# B&R Automation Studio project MIG1 (part 8)

#### UDP_Client.c - Init, cyclic, exit code
```c
#include <bur/plctypes.h>

#ifdef _DEFAULT_INCLUDES
	#include <AsDefault.h>
#endif
#include <..\GlobalDef.h>
#include <..\GlobalDecl.h>

#include <..\Lib\Statelib.c>
#include <..\Lib\LoggerLib.c>
#include <..\Lib\WSI_lib.c>

_LOCAL char TML_PLC_IP_Address[16];

typedef struct UDP_int_typ{

	UdpSend_typ send;
	UdpRecv_typ receive;
	UdpClose_typ close;
	UdpOpen_typ	open;

}UDP_int_typ;

typedef struct UDP_typ{

    UINT Step;

	UDINT SentCntr;
	UDINT RecevCntr;

	UDP_int_typ Intr;
	RS_Channel_typ *pSendChan;
	RS_Channel_typ *pRecevChan;

}UDP_typ;

_LOCAL UDP_typ UDP_Config[2];
_LOCAL UDP_typ UDP_Msg[2];

_LOCAL plcstring SrvIP[20];

_LOCAL UINT status;
_LOCAL plcbit sendNewMsg;
_LOCAL UINT receive_cntr;
_LOCAL UINT push_Cntr;

_LOCAL UINT ReceivedCntr;

_LOCAL plcstring KK_String[128];
_LOCAL USINT KK_Char;

_LOCAL plcbit firstScan;

void _INIT ProgramInit(void)
{UINT i;

	strcpy(SrvIP , "192.168.10.11");  // Must be Axis ID 10
	//strcpy(SrvIP , "192.168.19.11"); // This is default IP in new converter
	//strcpy(SrvIP , "255.255.255.255");

	//strcpy(TML_PLC_IP_Address , "192.168.11.123" ); // My PLC  Address - PowerLink Channel
	strcpy(TML_PLC_IP_Address , "192.168.10.123" ); // My PLC  Address - Ethernet Channel

	i = 0;
	// Initialize UDP open function block
	UDP_Config[i].Intr.open.enable = 0;
	UDP_Config[i].Intr.open.options = 0;
	UDP_Config[i].Intr.open.pIfAddr = (UDINT)&TML_PLC_IP_Address[0];
	UDP_Config[i].Intr.open.port = 30689;
	UDP_Config[i].Intr.open.ident = 0;

	// Initialize UDP send function block
	UDP_Config[i].Intr.send.enable = 0;
	UDP_Config[i].Intr.send.flags = 0;
	UDP_Config[i].Intr.send.pHost = (UDINT)&SrvIP[0];
	UDP_Config[i].Intr.send.port = 30689;

	UDP_Config[i].Intr.receive.ident = 0;
	UDP_Config[i].Intr.receive.enable = 1;
	UDP_Config[i].Intr.receive.pIpAddr = 0;
	UDP_Config[i].Intr.receive.flags = 0;

	// Initialize UDP open function block
	UDP_Msg[i].Intr.open.enable = 0;
	UDP_Msg[i].Intr.open.options = 0;
	UDP_Msg[i].Intr.open.pIfAddr = (UDINT)&TML_PLC_IP_Address[0];
	UDP_Msg[i].Intr.open.port = 1700;
	UDP_Msg[i].Intr.open.ident = 0;

	// Initialize UDP send function block
	UDP_Msg[i].Intr.send.enable = 0;
	UDP_Msg[i].Intr.send.flags = 0;
	UDP_Msg[i].Intr.send.pHost = (UDINT)&SrvIP[0];
	UDP_Msg[i].Intr.send.port = 1700;

	UDP_Msg[i].Intr.receive.ident = 0;
	UDP_Msg[i].Intr.receive.enable = 1;
	UDP_Msg[i].Intr.receive.flags = 0;
	UDP_Msg[i].Intr.receive.pIpAddr = 0;

	////////////////////////////////////////////////////
	UDP_Config[i].pRecevChan = &TML_Data_Chan[1];
	UDP_Config[i].pSendChan = &UDP_Connect_Send[i];

	UDP_Msg[i].pRecevChan = 0;
	UDP_Msg[i].pSendChan = &TML_Msg_Chan[1];

	////////////////////////
	//UDP_Config[i].Step = 1;
	//UDP_Msg[i].Step = 1;

	// Start Connection
	UDP_Config[i].pSendChan->Data[0] = 0x01;
	UDP_Config[i].pSendChan->Len = 1;

	UDP_Ready = 0;

	firstScan = 1;

	//Kick_TML_Cmd = 1;

}

void _CYCLIC ProgramCyclic(void)
{
UINT i , k ;

	//if(ESTOP && firstScan){
	if(firstScan){
		Kick_TML_Cmd = 1;
		firstScan = 0;

	}

	switch(Kick_TML_Cmd){

		case 1:

			UDP_Ready = 0;

			TML_mgr[0].hrdw[0].RXCount = 0;
			TML_mgr[0].hrdw[1].RXCount = 0;

			TML_mgr[1].hrdw[0].RXCount = 0;
			TML_mgr[1].hrdw[1].RXCount = 0;

			TML_mgr[0].hrdw[0].TXCount = 0;
			TML_mgr[0].hrdw[1].TXCount = 0;

			TML_mgr[1].hrdw[0].TXCount = 0;
			TML_mgr[1].hrdw[1].TXCount = 0;

			TML_mgr[0].hrdw[0].TXCountReadBack = TML_mgr[0].hrdw[0].TXCount;
			TML_mgr[0].hrdw[1].TXCountReadBack = TML_mgr[0].hrdw[1].TXCount;

			TML_mgr[1].hrdw[0].TXCountReadBack = TML_mgr[1].hrdw[0].TXCount;
			TML_mgr[1].hrdw[1].TXCountReadBack = TML_mgr[1].hrdw[1].TXCount;

			if(UDP_Config[0].Step == 10)
				UDP_Config[0].Step = 20;
			else
				UDP_Config[0].Step = 1;

			if(UDP_Msg[0].Step == 10)
				UDP_Msg[0].Step = 20;
			else
				UDP_Msg[0].Step = 1;

			Kick_TML_Cmd++;

		break;

		case 2:

			if((UDP_Msg[0].Step == 10)
				&& (UDP_Config[0].Step == 10)){

				UDP_Connect_Send[0].Cntr = 0;
				UDP_Connect_Send[0].Len = 1;

				Kick_TML_Cmd++;

			}

		break;

		case 3:

			if(UDP_Connect_Send[0].Cntr > 0)
				Kick_TML_Cmd++;

			Kick_TML_Cmd++;

		break;

		case 4:

			Kick_TML_Cmd++;

			TML_Msg_Chan[0].Trash_Cntr = 0;
			TML_Data_Chan[0].Trash_Cntr = 0;

			UDP_Ready = 1;

		break;

	}

	for(i = 0 ; i < 1 ; i++){

		for(k = 0 ; k < 2 ; k++){

			switch(k){

				case 0: 	UDP_Socket(&UDP_Config[i]);   	break;

				case 1: 	UDP_Socket(&UDP_Msg[i]);  		break;

			}

		}

	}

}

void UDP_Socket(UDP_typ *udp){

	switch(udp->Step){

			case 0:

			break;

			case 1:

				if(udp->pRecevChan){
					udp->Intr.receive.pData = (UDINT)&udp->pRecevChan->Data[0];
					udp->Intr.receive.datamax = 32;

				}else{
					udp->Intr.receive.pData = 0;
					udp->Intr.receive.datamax = 0;
				}

				if(udp->pSendChan){
					udp->Intr.send.pData = (UDINT)&udp->pSendChan->Data[0];
					udp->Intr.send.datalen = 0;
				}
				else{
					udp->Intr.send.pData = 0;
					udp->Intr.send.datalen = 0;
				}

				udp->Intr.open.enable = 1;

				UdpOpen(&udp->Intr.open);

				if(udp->Intr.open.ident && (udp->Intr.open.status == 0)){

					udp->Intr.send.enable = 1;
					udp->Intr.receive.enable = 1;

					udp->Intr.send.ident = udp->Intr.open.ident;
					udp->Intr.receive.ident = udp->Intr.open.ident;
					udp->Intr.close.ident = udp->Intr.open.ident;

					udp->Step = 10;

				}
				else if(udp->Intr.open.status == 32502){ // Port already opened

					udp->Intr.close.ident = udp->Intr.open.ident;
					udp->Intr.close.enable = 1;
					udp->Step = 20;
				}
				else if(udp->Intr.open.status != ERR_FUB_BUSY)
					udp->Step = 102;

			break;

			case 10:

				//////////////////////////////

				if(udp->pSendChan){

					if(udp->pSendChan->Len > 0){

						udp->Intr.send.datalen = udp->pSendChan->Len;
						UdpSend(&udp->Intr.send);

						if(udp->Intr.send.status == 0){

							udp->Intr.send.datalen = 0;

							udp->pSendChan->_len_prev = udp->pSendChan->Len;
							udp->pSendChan->Len = 0;
							udp->SentCntr++;
							udp->pSendChan->Cntr++;
						}
						else if(udp->Intr.send.status != ERR_FUB_BUSY){

							udp->Intr.send.datalen = 0;

						 	udp->pSendChan->_len_prev = udp->pSendChan->Len;
							udp->pSendChan->Len = 0;
							udp->Step = 110;
						}
					}

				}

				//////////////////////////////////////////////////////////////////

				if(udp->pRecevChan){

					if((udp->pRecevChan->Len == 0)
						&& (udp->pSendChan->Len == 0)){

						UdpRecv(&udp->Intr.receive);

						if(udp->Intr.receive.status == ERR_FUB_BUSY)
						{  }// Process busy

						else if(udp->Intr.receive.status == 0)/* Data received */
						{
							udp->pRecevChan->Len = udp->Intr.receive.recvlen;
							udp->RecevCntr++;
							udp->pRecevChan->Cntr++;

						}
						else if(udp->Intr.receive.status != 32505) // Error ( 32505 is no datat received)
							udp->Step = 115;

					}
				}

			break;

			case 20:

				UdpClose(&udp->Intr.close);

				if(udp->Intr.close.status == ERR_FUB_BUSY)
				{  }// Process busy

				else if(udp->Intr.close.status) {// error
						//udp->Step = 120;
						udp->Step = 1;
				}
				else{

					udp->Intr.open.ident = 0;
					udp->Intr.send.ident = 0;
					udp->Intr.close.ident = 0;
					udp->Intr.receive.ident = 0;

					udp->Step = 1;
				}

			break;

			case 101:
			case 102:
			case 110:
			case 115:
			case 120:

			break;

		}

}
```

### Program Logical/Calibr (ANSIC)

#### Clibr.c - Init, cyclic, exit code
```c
#include <bur/plctypes.h>

#ifdef _DEFAULT_INCLUDES
	#include <AsDefault.h>
#endif

#include <..\GlobalDef.h>
#include <..\GlobalDecl.h>

_LOCAL SINT TVL_Calibr_Cmd;
_LOCAL USINT TVL_Calibr_Step;
_LOCAL TON_typ TVL_Calibr_Tmr;

void _INIT ProgramInit(void)
{

}

void _CYCLIC ProgramCyclic(void)
{

}

void _EXIT ProgramExit(void)
{

}
```

### Program Logical/LincolnPS (ANSIC)

#### LincolnPS.c - Cyclic code
```c
///   ARC Link address: "192.168.10.2"

#include <bur/plctypes.h>

#ifdef _DEFAULT_INCLUDES
	#include <AsDefault.h>
#endif

#include <..\Lib\utilityLib\bgdebug.h>

#include <..\Lib\libUDP\libUDP.h>
#include <..\Lib\libUDP\libUDP.c>

#include <..\Lib\arclink\arclink.h>
#include <..\Lib\arclink\arclink.c>

#define REC_BUF_LEN 	512
#define REC_NUM 	8
#define ARCCOM_TIMEOUT 2000

_GLOBAL Arc_Link_typ ArcLink;

/*
#define REC_BUF_LEN 	4+1
#define REC_NUM 	4
*/

USINT send_data[REC_BUF_LEN];
USINT receive_data[REC_BUF_LEN];
USINT temp_data[REC_BUF_LEN * 3];

_LOCAL RingBuffer RingBufIn;
_LOCAL RingBuffer RingBufOut;
char RingBufInData[(REC_BUF_LEN +4) * REC_NUM];
char RingBufOutData[(REC_BUF_LEN +4) * REC_NUM];
char MsgInData[REC_BUF_LEN];
char MsgOutData[REC_BUF_LEN];

_LOCAL Arc_Link_typ *arcLink;
_LOCAL UDP_typ2 ArcLink_UDP;
_LOCAL plcbit Run_DispatchOutgoingMessages;

_LOCAL char ArcLinkPS_IP_Address[16];
_LOCAL char ArcLinkPLC_IP_Address[16];
_LOCAL plcbit ArcLink_Run;

_LOCAL plcbit KK_ReadParamData;

/*
_LOCAL plcbit RunOutgoingDispatcher;

/// Test Ring Buffer

_LOCAL plcbit KK_Write , KK_Read;
_LOCAL plcstring KK_text_Write[32] ,  KK_text_Read[32];
_LOCAL UDINT KK_Write_Len , KK_Read_Len;
_LOCAL plcbit KK_isEmpty , KK_isFULL;

_LOCAL plcbit K_Send_Req_Action_28 , K_Send_Resp_Action_28;

const char Action_28_Request[29] = {
	0x00, 0x02, 0x0a, 0x4a, 0x00, 0x00, 0x00, 0x00, 0x00, 0x13,
	0x00, 0x32, 0x08, 0x00, 0x00, 0x01, 0x02, 0x01, 0x00, 0x16,
	0x00, 0x00, 0x00, 0xff, 0x01, 0xfe, 0x01, 0x00, 0x01,
};

const char Action_28_Respond[16] = {
	0x00, 0x03, 0x0A, 0x4A, 0x00, 0x00, 0x00, 0x00, 0x00, 0x06,
	0x01, 0x00, 0x00, 0x06, 0x00, 0x00,

};

*/

////////////////////////////////////////////

//UDP Receive Callback function to push data on ring buffer
static void udpReceivedNewData(UDINT pRxBuffer, UDINT RxDataLen , UDINT ringBuf){

	DBG("New Data Received  of Length %d \r\n" , RxDataLen);

	ckConvertByteStreamToHex(pRxBuffer, temp_data, RxDataLen, sizeof(temp_data));
	DBG("(Hex): %s  \r\n" , temp_data);

	if(ringBuf){

		if(!RingBuffer_isFull((RingBuffer*) ringBuf))
			RingBuffer_writeRecord((RingBuffer*) ringBuf, pRxBuffer, RxDataLen);

	}

}
//UDP Transmit Callback function for debugging purpose
static void udpTransmitedNewData(UDINT pTxBuffer, UDINT pTxDataLen){

	DBG("New Data Trasmitted of Length %d  \r\n " , pTxDataLen );
	ckConvertByteStreamToHex(pTxBuffer, temp_data, pTxDataLen, sizeof(temp_data));
	DBG("(Hex): %s  \r\n" , temp_data);

}

//handle network timeout
void ArcLink_Timer(Arc_Link_typ *arc);

//handle error/status interface
void error_status_handler(Arc_Link_typ *arc);

void _INIT ProgramInit(void){
Arc_Link_typ *arc;
UDP_typ2 *udp;

	//ArcLink.robot.Comm.CntrlParamReq.Attribute_ID = 517;
	ArcLink.robot.Comm.CntrlParamReq.Attribute_ID = 0;
	ArcLink.robot.Comm.CntrlParamReq.Weld_Mode = 200;

	/*
	Work-point	517 Primary control.
	Trim	518 Arc length control (typically).
	Wave-Control 1	519 Process adjustment.
	Wave-Control 2	520 Process adjustment.
	Wave-Control 3	521 Process adjustment.
	Wave-Control 4	522 Process adjustment.
	*/

	ArcLink_Run = 1;

	strcpy(ArcLinkPS_IP_Address , "192.168.10.2" );
	//strcpy(ArcLinkPS_IP_Address , "192.168.1.2" ); // Przez PowerLink Module

	strcpy(ArcLinkPLC_IP_Address , "192.168.10.123" ); // My PLC  Address

	Run_DispatchOutgoingMessages = 1;

	udp = &ArcLink_UDP;

	//if(!arcLink)
		//arcLink = ArcLink_init(REC_NUM , REC_BUF_LEN );

	arcLink = &ArcLink;

	if(arcLink){
		udp->listener_config.port = 4323;
		udp->listener_config.buffer = receive_data;
		udp->listener_config.bufferSize = REC_BUF_LEN;
		udp->listener.iRxCallback = (UDINT)udpReceivedNewData;
		//udp->listener.iRxRingBuf = arcLink->bufIN;
		udp->listener.iRxRingBuf = (UDINT)&RingBufIn;

		//strcpy(udp->send.iIPaddress , "192.168.10.2");
		//	strcpy(udp->send.iIPaddress , "192.168.36.88");
		//strcpy(udp->send.iIPaddress , "192.168.10.178");
		udp->send.iPort = 4323;
		udp->send.iBuffer = send_data;
		udp->send.iBufferSize = REC_BUF_LEN;
		udp->send.iTxCallback = (UDINT)udpTransmitedNewData;

		udp->internal.UdpOpen_0.pIfAddr = (UDINT)&ArcLinkPLC_IP_Address[0];

	}
}

void _CYCLIC ProgramCyclic(void){

UDP_typ2 *udp;

	udp = &ArcLink_UDP;

	if(!arcLink)
		return;

	if(!RingBufIn.buffer)
		RingBuffer_Init(&RingBufIn , &RingBufInData , REC_NUM , REC_BUF_LEN);

	if(!RingBufOut.buffer)
		RingBuffer_Init(&RingBufOut , &RingBufOutData , REC_NUM , REC_BUF_LEN);

	if(!arcLink->bufIN
		|| !arcLink->bufOUT
		|| !arcLink->internal.pInMsg
		|| !arcLink->internal.pOutMsg)
	ArcLink_init(arcLink , &RingBufIn, &RingBufOut, MsgInData  , MsgOutData, REC_BUF_LEN );

	//////////////////////////////////////
	if(Run_DispatchOutgoingMessages){

		if(!RingBuffer_isEmpty(arcLink->bufOUT) && !udp->send.iSendCMD){

			udp->send.iBufferSize = RingBuffer_readRecord(arcLink->bufOUT, udp->send.iBuffer);
			udp->send.iSendCMD = 1;

		}

	}

	if((strlen(ArcLinkPS_IP_Address) > 0) && ArcLink_Run) {

		if(udp->internal.step == 0)
			strcpy(udp->send.iIPaddress , ArcLinkPS_IP_Address);

		Udp_cyclic(udp);
		ArcLink_cyclic(arcLink);

	}

	 if(KK_ReadParamData){

	 	KK_ReadParamData = 0;

		ArcLink.robot.Intrf.xCMD = ROBOT_READ_WC_PARAM_DATA;
		ArcLink.robot.Comm.CntrlParamReq.Attribute_ID++;
		if(ArcLink.robot.Comm.CntrlParamReq.Attribute_ID  < 517)
			ArcLink.robot.Comm.CntrlParamReq.Attribute_ID  = 517;
		else if(ArcLink.robot.Comm.CntrlParamReq.Attribute_ID  > 522)
			ArcLink.robot.Comm.CntrlParamReq.Attribute_ID  = 522;

	 }
}
```

### Program Logical/LocalJog (ANSIC)

#### LocalJog.c - Init, cyclic, exit code
```c
#include <bur/plctypes.h>

#ifdef _DEFAULT_INCLUDES
	#include <AsDefault.h>
#endif

#include <..\GlobalDef.h>
#include <..\GlobalDecl.h>

#include <..\Lib\Statelib.c>
#include <..\Lib\LoggerLib.c>
#include <..\Lib\WSI_lib.c>

_LOCAL TON_typ JogMode_Tmr;
_LOCAL float ModeTmo;

_LOCAL plcbit SetLED;

_LOCAL USINT _LocalJogMode;
USINT JogFwdRev(plcbit fwd , plcbit rev);
void LED_Step_Seq();

_LOCAL BOOL blink , _blink;
BOOL _blink;
_LOCAL UINT blinkOnTmr , blinkOffTmr;

_LOCAL TON_typ LED_Tmr;
_LOCAL UINT LED_Indx , LED_Step ;
UINT _LED_Indx;

_LOCAL plcbit LED_Static_Style;

plcbit _Remote_SW;
plcbit _SR_Done;
plcbit _LocalJog_FWD , _LocalJog_REV;

USINT _indx_Limit_Bypass_Btn;

_LOCAL plcbit HMI_INDX_Inp2 , HMI_INDX_Inp3 , HMI_INDX_Out2;

_LOCAL plcbit KK_Block_LED , KK_AllowAll_LED;
_LOCAL float KK_Blink;

void _INIT ProgramInit(void)
{

	KK_Block_LED = 0;
	KK_AllowAll_LED = 0;
	KK_Blink = 0.5;

	Head.Remote_SW = 1;
	ModeTmo = 15.0;

	HardwInit_Done = 0;
	LED_Static_Style = 1;

	Glbl_TML_CMD_Delay = Glbl_TML_CMD_Delay;
}

void _CYCLIC ProgramCyclic(void)
{

USINT tml_indx ;

/*
#define MODE_NONE 	0
#define MODE_TVL 	1
#define MODE_OSC 	2
#define MODE_AHC 	3
#define MODE_WF 	4
#define MODE_INDX 	5

TravelJog.IN
OSCJog_Cmd
AHCJog.IN
WFJog.IN
IndexJog.IN

*/

/** Blink **/
if(blinkOnTmr++ < 150)		blink = 1;
else if(blinkOffTmr++ < 300)	blink = 0;
else{ blinkOnTmr = 0; blinkOffTmr = 0;}

////////////////////////////////////////////////////////
if(HardwReady){

	if(!HardwInit_Done){
		LED_Step = 0;
		LED_CMD = 20;
		_Remote_SW = Head.Remote_SW;
	}

	HardwInit_Done = 1;

}

if(HardwInit_Done && HardwReady){

	Head.Remote_SW = !TML_MTR_INST[TML_AX_WF].DigInp[1];
	//Head.Remote_SW = 1;

	Head.LocalJog_FWD = !TML_MTR_INST[TML_AX_OSC].DigInp[1];
	Head.LocalJog_REV = !TML_MTR_INST[TML_AX_OSC].DigInp[0];

	if(LocalJogMode != MODE_NONE){

		if(Head.LocalJog_FWD || Head.LocalJog_REV)
			TimerStart(&JogMode_Tmr, ModeTmo);

	}

	if((Seq.State > 0) && (Seq.State < 25))
			TimerStart(&JogMode_Tmr, ModeTmo);

	if(!TML_MTR_INST[TML_AX_TVL].DigInp[0]){
		LocalJogMode = MODE_TVL;
		TimerStart(&JogMode_Tmr, ModeTmo);
	}

	else if(!TML_MTR_INST[TML_AX_INDX_EXT].DigInp[1]){
		LocalJogMode = MODE_OSC;
		TimerStart(&JogMode_Tmr, ModeTmo);
	}

	else if(!TML_MTR_INST[TML_AX_TVL].DigInp[1]){
		LocalJogMode = MODE_AHC;
		TimerStart(&JogMode_Tmr, ModeTmo);
	}

	else if(!TML_MTR_INST[TML_AX_INDX].DigInp[1]){
		LocalJogMode = MODE_WF;
		TimerStart(&JogMode_Tmr, ModeTmo);
	}

	else if(!TML_MTR_INST[TML_AX_INDX].DigInp[0] && (!MachCfg.IndxExt)){
		LocalJogMode = MODE_INDX;
		TimerStart(&JogMode_Tmr, ModeTmo);
	}

	else if(!TML_MTR_INST[TML_AX_INDX_EXT].DigInp[0] && (MachCfg.IndxExt)){
		LocalJogMode = MODE_INDX_EXT;
		TimerStart(&JogMode_Tmr, ModeTmo);
	}

	else if(TimerIsTimeOut(&JogMode_Tmr) && (OSC_Step != 10))
		LocalJogMode = MODE_NONE;

}
else {

	Head.Remote_SW = 0;
	Head.LocalJog_FWD = 0;
	Head.LocalJog_REV = 0;

	return;

}

	if(Head.Remote_SW)
		LocalJogMode = MODE_NONE;

	if(Head.Remote_SW && !_Remote_SW)
		//LED_CMD = 40;
		LED_CMD = 10;
	else if(!Head.Remote_SW && _Remote_SW)
		//LED_CMD = 30;
		LED_CMD = 20;

/*
	if(Head.Remote_SW != _Remote_SW){

		OSCJog = Stop;

		OSCJog_Cmd = Stop;

		TravelJog.IN = Stop;

		AHCJog.IN = Stop;

		WFJog.IN = Stop;

		IndexJog.IN = Stop;

	}
	*/

	_Remote_SW = Head.Remote_SW;

//////////  Override POT & NOT on INDX motor

	/*
	if(Head.Remote_SW || !HardwInit_Done || (AccessLevel < 0)){

		INDX_Limit_Bypass_Btn = 0;
		_indx_Limit_Bypass_Btn = INDX_Limit_Bypass_Btn;

	}
	*/

	if(MachCfg.IndxExt)
		tml_indx = TML_AX_INDX_EXT;
	else
		tml_indx = TML_AX_INDX;

	HMI_INDX_Inp2 = TML_MTR_INST[tml_indx].DigInp[2];
	HMI_INDX_Inp3 = TML_MTR_INST[tml_indx].DigInp[3];

	HMI_INDX_Out2 = TML_MTR_INST[tml_indx].DigOut_stat[2];

	if(INDX_Limit_Bypass_Btn && !_indx_Limit_Bypass_Btn){

		if(TML_MTR_INST[tml_indx].xCMD == TML_IDLE){
				TML_MTR_INST[tml_indx].xCMD 	= TML_RST_OUT3_CMD;

			_indx_Limit_Bypass_Btn = INDX_Limit_Bypass_Btn;

		}

	}
	else if(!INDX_Limit_Bypass_Btn && _indx_Limit_Bypass_Btn){

		if(TML_MTR_INST[tml_indx].xCMD == TML_IDLE){
				TML_MTR_INST[tml_indx].xCMD 	= TML_SET_OUT3_CMD;

			_indx_Limit_Bypass_Btn = INDX_Limit_Bypass_Btn;

		}

	}

/////////////////////////////////////////////////////////

	switch(LocalJogMode){

		case MODE_TVL:

			TravelJog.IN = JogFwdRev(Head.LocalJog_FWD , Head.LocalJog_REV);

			if(_LocalJogMode != LocalJogMode)
				LED_CMD = 11;

		break;

		case MODE_OSC:
			 // (0, 1 ,-1)

			if(TML_MTR_INST[TML_AX_INDX_EXT].DigInp[1]){

				if(HardwReady && !Head.Remote_SW){

					if(Head.LocalJog_REV  && !_LocalJog_REV )
						//OSCToggle = 1;
						OSCToggle = !OSCToggle;

					else if(Head.LocalJog_FWD  && !_LocalJog_FWD ){
						if(OSC_Step == 5)
							OSCJog = 1;
						else if(OSC_Step == 10)
							OSCJog = 0;
					}

				}

			}
			else{

				if(Head.LocalJog_FWD == Head.LocalJog_REV)
					OSCJog_Cmd = 0;

				else if(Head.LocalJog_FWD){

					/*
					if(OSCJog)
						OSCJog = 0;
					else */
						OSCJog_Cmd = 1;
				}
				else {
					/*
					if(OSCJog)
						OSCJog = 0;
					else */
						OSCJog_Cmd = -1;
				}
			}

			if(_LocalJogMode != LocalJogMode)
				LED_CMD = 14;

		break;

		case MODE_AHC:

			AHCJog.IN = JogFwdRev(Head.LocalJog_FWD , Head.LocalJog_REV);
			if(_LocalJogMode != LocalJogMode)
				LED_CMD = 13;

		break;

		case MODE_WF:

			WFJog.IN = JogFwdRev(Head.LocalJog_FWD , Head.LocalJog_REV);

			if(_LocalJogMode != LocalJogMode)
				LED_CMD = 15;

		break;

		case MODE_INDX:

			IndexJog.IN = JogFwdRev(Head.LocalJog_FWD , Head.LocalJog_REV);
			if(_LocalJogMode != LocalJogMode)
				LED_CMD = 12;

		break;

		case MODE_INDX_EXT:

			//IndexExtJog.IN = JogFwdRev(Head.LocalJog_FWD , Head.LocalJog_REV);
			IndexJog.IN = JogFwdRev(Head.LocalJog_FWD , Head.LocalJog_REV);
			if(_LocalJogMode != LocalJogMode)
				LED_CMD = 16;

		break;

		default:

			 if (_LocalJogMode != LocalJogMode){

				if(LED_Static_Style)
					LED_CMD = 20;
				else
					LED_CMD = 30;

			 	OSCJog = Stop;

				OSCJog_Cmd = Stop;

				TravelJog.IN = Stop;

				AHCJog.IN = Stop;

				WFJog.IN = Stop;

				IndexJog.IN = Stop;

			}
			 /*
			 else if(HardwReady && !Head.Remote_SW){

				if(Head.LocalJog_FWD && Head.LocalJog_REV && !_LocalJog_FWD_REV )
					OSCToggle = !OSCToggle;

			}
			*/

		break;

	}

	if(_LocalJogMode != LocalJogMode)
		OSCJog = 0;

	_LocalJog_FWD = (Head.LocalJog_FWD);
	_LocalJog_REV = (Head.LocalJog_REV);

	_LocalJogMode = LocalJogMode;
	_blink = blink;
	TimerExecute(&JogMode_Tmr);

	if(LED_CMD){

		TimerStart(&LED_Tmr,0.02);

		if(LED_CMD == 255){ // Reset

			LED_Step = 0;
			LED_Indx = 1;
			LED_CMD = 0;

		}
		else if(LED_CMD <= 10){

			if((LED_Indx > 6)
				|| (LED_Indx == 0))
				LED_Indx = 1;

			LED_Step = LED_CMD;

		}
		else if(LED_CMD < 20){	// Imprtant - Clear & Set

			if((LED_Indx > 6)
			|| (LED_Indx == 0))
				LED_Indx = 1;

			LED_Step = 10;

		}
		else if(LED_CMD == 20){
			LED_Step = 20;
			LED_Indx = 1;
			LED_CMD = 0;

		}
		else if(LED_CMD == 30){
			LED_Step = 30;
			LED_Indx = 1;
			LED_CMD = 0;

		}
		else if(LED_CMD == 40){
			LED_Step = 40;
			LED_Indx = 1;
			LED_CMD = 0;
		}
		else if(LED_CMD == 100){

			if(LED_Step < 100)
				LED_Step = 100;

			LED_CMD = 0;

		}

		else {

			LED_Step = 20;
			LED_CMD = 0;
		}

	}

	if(LED_One_Blink_Req || (Seq.State == 0) || (Seq.State > 25) || KK_AllowAll_LED){

		if(!KK_Block_LED)
			LED_Step_Seq();

	}

	TimerExecute(&LED_Tmr);

}

USINT JogFwdRev(plcbit fwd , plcbit rev){
USINT ret;
// Stop , Reverse , Forward

	if(fwd == rev)
		ret = Stop;
	else if(fwd)
		ret = Forward;
	else if(rev)
		ret = Reverse;
	else
		ret = Stop;

	return ret;

}

void LED_Step_Seq(){

switch(LED_Step){

		case 0:

	/*
	TML_MTR_INST[TML_AX_TVL].xCMD	= TML_SET_OUT1_CMD; // TVL
	TML_MTR_INST[TML_AX_WF].xCMD	= TML_SET_OUT4_CMD; // OUT4 INDX
	TML_MTR_INST[TML_AX_AHC].xCMD	= TML_SET_OUT0_CMD; // AHC
	TML_MTR_INST[TML_AX_OSC].xCMD	= TML_SET_OUT0_CMD; // OSC
	TML_MTR_INST[TML_AX_WF].xCMD	= TML_SET_OUT1_CMD; // WF
	TML_MTR_INST[TML_AX_TVL].xCMD	= TML_SET_OUT4_CMD; // EXT INDX

	TML_SET_OUT1_CMD  		VECT_Rst_OUT1
	*/

		break;

		//////////////////////////////////////////////////////////////////////////////////////

		case 1:

			if(!VectorStateMach[VECT_AX_TVL].xCmd_busy){
				VectorStateMach[VECT_AX_TVL].xCMD 	= VECT_Set_OUT1; // TVL
				LED_CMD = 0;
				LED_Step = 0;

			}
		break;

		case 2:

			if(!VectorStateMach[VECT_AX_WF].xCmd_busy){
				VectorStateMach[VECT_AX_WF].xCMD 	= VECT_Set_OUT4; // OUT4 INDX
				LED_CMD = 0;
				LED_Step = 0;

			}
		break;

		case 3:

			if(!VectorStateMach[VECT_AX_AHC].xCmd_busy){
				VectorStateMach[VECT_AX_AHC].xCMD 	= VECT_Set_OUT0; // AHC
				LED_CMD = 0;
				LED_Step = 0;

			}
		break;

		case 4:

			if(!VectorStateMach[VECT_AX_OSC].xCmd_busy){
				VectorStateMach[VECT_AX_OSC].xCMD 	= VECT_Set_OUT0; // OSC
				LED_CMD = 0;
				LED_Step = 0;

			}
		break;

		case 5:

			if(!VectorStateMach[VECT_AX_WF].xCmd_busy){
				VectorStateMach[VECT_AX_WF].xCMD 	= VECT_Set_OUT1; // WF
				LED_CMD = 0;
				LED_Step = 0;

			}
		break;

		case 6:

			if(!VectorStateMach[VECT_AX_TVL].xCmd_busy){
				VectorStateMach[VECT_AX_TVL].xCMD 	= VECT_Set_OUT4; // EXT INDX
				LED_CMD = 0;
				LED_Step = 0;

			}
		break;

		//****/

		case 10:

			switch(LED_Indx){

				case 1:

					if(!VectorStateMach[VECT_AX_TVL].xCmd_busy){

						VectorStateMach[VECT_AX_TVL].xCMD 	= VECT_Rst_OUT1; // TVL
						//
						LED_Indx++;
					}

				break;

				case 2:

					if(!VectorStateMach[VECT_AX_WF].xCmd_busy){

						VectorStateMach[VECT_AX_WF].xCMD 	= VECT_Rst_OUT4; // OUT4 INDX
						//
						LED_Indx++;
					}

				break;

				case 3:

					if(!VectorStateMach[VECT_AX_AHC].xCmd_busy){
						VectorStateMach[VECT_AX_AHC].xCMD 	= VECT_Rst_OUT0; // AHC
						//
						LED_Indx++;
					}

				break;

				case 4:

					if(!VectorStateMach[VECT_AX_OSC].xCmd_busy){
						VectorStateMach[VECT_AX_OSC].xCMD 	= VECT_Rst_OUT0; // OSC
						//
						LED_Indx++;
					}

				break;

				case 5:

					if(!VectorStateMach[VECT_AX_WF].xCmd_busy){
						VectorStateMach[VECT_AX_WF].xCMD 	= VECT_Rst_OUT1; // WF
						//
						LED_Indx++;
					}

				break;

				case 6:

					if(!VectorStateMach[VECT_AX_TVL].xCmd_busy){
						VectorStateMach[VECT_AX_TVL].xCMD 	= VECT_Rst_OUT4; // EXT INDX
						//
						LED_Indx++;
					}

				break;

				default:

					LED_Indx = 0;

				break;
			}

			if(LED_Indx > 6) {// Done

				if(Head.Remote_SW)
					LED_Step = 40;
				else
					LED_Step = LED_CMD%10;

				LED_CMD = 0;

			}

		break;

		///////////////////////////////////////////////////////////////////////////////

		case 20:

			switch(LED_Indx){

				case 1:

					if(!VectorStateMach[VECT_AX_TVL].xCmd_busy){

						VectorStateMach[VECT_AX_TVL].xCMD 	= VECT_Set_OUT1; // TVL
						//
						LED_Indx++;
					}

				break;

				case 2:

					if(!VectorStateMach[VECT_AX_WF].xCmd_busy){

						VectorStateMach[VECT_AX_WF].xCMD 	= VECT_Set_OUT4; // OUT4 INDX
						//
						LED_Indx++;
					}

				break;

				case 3:

					if(!VectorStateMach[VECT_AX_AHC].xCmd_busy){
						VectorStateMach[VECT_AX_AHC].xCMD 	= VECT_Set_OUT0; // AHC
						//
						LED_Indx++;
					}

				break;

				case 4:

					if(!VectorStateMach[VECT_AX_OSC].xCmd_busy){
						VectorStateMach[VECT_AX_OSC].xCMD 	= VECT_Set_OUT0; // OSC
						//
						LED_Indx++;
					}

				break;

				case 5:

					if(!VectorStateMach[VECT_AX_WF].xCmd_busy){
						VectorStateMach[VECT_AX_WF].xCMD 	= VECT_Set_OUT1; // WF
						//
						LED_Indx++;
					}

				break;

				case 6:

					if(!VectorStateMach[VECT_AX_TVL].xCmd_busy){
						VectorStateMach[VECT_AX_TVL].xCMD 	= VECT_Set_OUT4; // EXT INDX
						//
						LED_Indx++;
					}

				break;

				default:

					LED_Indx = 0;

				break;
			}

			if(LED_Indx > 6){ // Done
				LED_CMD = 0;

				if(LED_Static_Style)
					LED_Step = 0;
				else
					LED_Step = 30;

			}

		break;

		///////////////////////////////////////////////////////////////////////////////

		case 30:

				LED_CMD = 0;
				LED_Indx = 1;
				TimerStart(&LED_Tmr, 0.01);
				_SR_Done = 0;
				LED_Step++;

		break;

		case 31:

			if(LED_CMD)
				LED_Step = 0;

			if(!TimerIsTimeOut(&LED_Tmr))
				break;

			switch(LED_Indx){

				case 1:

					if(!VectorStateMach[VECT_AX_TVL].xCmd_busy){
						VectorStateMach[VECT_AX_TVL].xCMD 	= VECT_Rst_OUT1; // TVL
						_SR_Done = 1;
					}

				break;

				case 2:

					if(!VectorStateMach[VECT_AX_WF].xCmd_busy){
						VectorStateMach[VECT_AX_WF].xCMD 	= VECT_Rst_OUT4; // OUT4 INDX
						_SR_Done = 1;
					}

				break;

				case 3:
					if(!VectorStateMach[VECT_AX_AHC].xCmd_busy){
						VectorStateMach[VECT_AX_AHC].xCMD 	= VECT_Rst_OUT0; // AHC
						_SR_Done = 1;
					}

				break;

				case 4:

					if(!VectorStateMach[VECT_AX_OSC].xCmd_busy){
						VectorStateMach[VECT_AX_OSC].xCMD 	= VECT_Rst_OUT0; // OSC
						_SR_Done = 1;
					}

				break;

				case 5:

					if(!VectorStateMach[VECT_AX_WF].xCmd_busy){
						VectorStateMach[VECT_AX_WF].xCMD 	= VECT_Rst_OUT1; // WF
						_SR_Done = 1;
					}

				break;

				case 6:

					if(!VectorStateMach[VECT_AX_TVL].xCmd_busy){
						VectorStateMach[VECT_AX_TVL].xCMD 	= VECT_Rst_OUT4; // EXT INDX
						_SR_Done = 1;
					}

				break;

				default:

					LED_Indx = 0;

				break;
			 }
			if(_SR_Done){
				_SR_Done = 0;
				TimerStart(&LED_Tmr, KK_Blink * 0.5);
				LED_Indx++;
				if(LED_Indx > 6){
					LED_Indx = 1;
					TimerStart(&LED_Tmr, KK_Blink *0.5);
					LED_Step++;
				}

			}

		break;

		case 32:

			if(!TimerIsTimeOut(&LED_Tmr))
				break;

			switch(LED_Indx){

				case 1:
					if(!VectorStateMach[VECT_AX_TVL].xCmd_busy){
						VectorStateMach[VECT_AX_TVL].xCMD 	= VECT_Set_OUT1; // TVL
						_SR_Done = 1;
					}

				break;

				case 2:

					if(!VectorStateMach[VECT_AX_WF].xCmd_busy){
						VectorStateMach[VECT_AX_WF].xCMD 	= VECT_Set_OUT4; // OUT4 INDX
						_SR_Done = 1;
					}

				break;

				case 3:

					if(!VectorStateMach[VECT_AX_AHC].xCmd_busy){
						VectorStateMach[VECT_AX_AHC].xCMD 	= VECT_Set_OUT0; // AHC
						_SR_Done = 1;
					}

				break;

				case 4:

					if(!VectorStateMach[VECT_AX_OSC].xCmd_busy){
						VectorStateMach[VECT_AX_OSC].xCMD 	= VECT_Set_OUT0; // OSC
						_SR_Done = 1;
					}

				break;

				case 5:

					if(!VectorStateMach[VECT_AX_WF].xCmd_busy){
						VectorStateMach[VECT_AX_WF].xCMD 	= VECT_Set_OUT1; // WF
						_SR_Done = 1;
					}

				break;

				case 6:

					if(!VectorStateMach[VECT_AX_TVL].xCmd_busy){
						VectorStateMach[VECT_AX_TVL].xCMD 	= VECT_Set_OUT4; // EXT INDX
						_SR_Done = 1;
					}

				break;

				default:

					LED_Indx = 0;

				break;
			 }

			if(_SR_Done){
				_SR_Done = 0;
				TimerStart(&LED_Tmr, KK_Blink *0.5);
				LED_Indx++;
				if(LED_Indx > 6){
					LED_Indx = 1;
					TimerStart(&LED_Tmr, KK_Blink *0.5);
					LED_Step = 31;
				}

			}

		break;

		case 33:

			if(LED_CMD)
				LED_Step = 0;

			if(!TimerIsTimeOut(&LED_Tmr))
				break;

			switch(LED_Indx){

				case 1:

					if((!VectorStateMach[VECT_AX_TVL].xCmd_busy)){

						VectorStateMach[VECT_AX_TVL].xCMD 	= VECT_Set_OUT1; // TVL
						_SR_Done = 1;
						LED_Indx++;
					}

				break;

				case 2:

					if((!VectorStateMach[VECT_AX_WF].xCmd_busy)){

						VectorStateMach[VECT_AX_WF].xCMD 	= VECT_Set_OUT4; // OUT4 INDX
						_SR_Done = 1;
						LED_Indx++;
					}

				break;

				case 3:

					if((!VectorStateMach[VECT_AX_AHC].xCmd_busy)){
						VectorStateMach[VECT_AX_AHC].xCMD 	= VECT_Set_OUT0; // AHC
						_SR_Done = 1;
						LED_Indx++;
					}

				break;

				case 4:

					if((!VectorStateMach[VECT_AX_OSC].xCmd_busy)){
						VectorStateMach[VECT_AX_OSC].xCMD 	= VECT_Set_OUT0; // OSC
						_SR_Done = 1;
						LED_Indx++;
					}

				break;

				case 5:

					if((!VectorStateMach[VECT_AX_WF].xCmd_busy)){
						VectorStateMach[VECT_AX_WF].xCMD 	= VECT_Set_OUT1; // WF
						_SR_Done = 1;
						LED_Indx++;
					}

				break;

				case 6:

					if((!VectorStateMach[VECT_AX_TVL].xCmd_busy)){
						VectorStateMach[VECT_AX_TVL].xCMD 	= VECT_Set_OUT4; // EXT INDX
						_SR_Done = 1;
						LED_Indx++;
					}

				break;

				default:

					LED_Indx = 0;

				break;
			}

			if(LED_Indx > 6){

				LED_Indx = 1;
			}

			if(_SR_Done){
				_SR_Done = 0;
				TimerStart(&LED_Tmr, KK_Blink *0.5);
				LED_Step = 31;

			}

		break;

		//////////////////////////////////////////////////////////////////////

		case 40:

			LED_CMD = 0;
			LED_Indx = 1;
			TimerStart(&LED_Tmr, 0.1);
			_SR_Done = 0;
			LED_Step++;

		break;

		case 41:

			if(LED_CMD)
				LED_Step = 0;

			if(!TimerIsTimeOut(&LED_Tmr))
				break;

			switch(LED_Indx){

				case 1:

					if(!VectorStateMach[VECT_AX_TVL].xCmd_busy){

						VectorStateMach[VECT_AX_TVL].xCMD	= VECT_Set_OUT1; // TVL
						_SR_Done = 1;
					}

				break;

				case 2:

					if(!VectorStateMach[VECT_AX_WF].xCmd_busy){

						VectorStateMach[VECT_AX_WF].xCMD	= VECT_Set_OUT4; // OUT4 INDX
						_SR_Done = 1;
					}

				break;

				case 3:

					if(!VectorStateMach[VECT_AX_AHC].xCmd_busy){
						VectorStateMach[VECT_AX_AHC].xCMD	= VECT_Set_OUT0; // AHC
						_SR_Done = 1;
					}

				break;

				case 4:

					if(!VectorStateMach[VECT_AX_OSC].xCmd_busy){
						VectorStateMach[VECT_AX_OSC].xCMD	= VECT_Set_OUT0; // OSC
						_SR_Done = 1;
					}

				break;

				case 5:

					if(!VectorStateMach[VECT_AX_WF].xCmd_busy){
						VectorStateMach[VECT_AX_WF].xCMD	= VECT_Set_OUT1; // WF
						_SR_Done = 1;
					}

				break;

				case 6:

					if(!VectorStateMach[VECT_AX_TVL].xCmd_busy){
						VectorStateMach[VECT_AX_TVL].xCMD	= VECT_Set_OUT4; // EXT INDX
						_SR_Done = 1;
					}

				break;

				default:

					LED_Indx = 0;

				break;
			 }
			if(_SR_Done){
				_SR_Done = 0;
				TimerStart(&LED_Tmr, KK_Blink);
				LED_Step++;

			}

		break;

		case 42:

			if(LED_CMD)
				LED_Step = 0;

			if(!TimerIsTimeOut(&LED_Tmr))
				break;

			switch(LED_Indx){

				case 1:

					if(TML_MTR_INST[TML_AX_TVL].Error){

						VectorStateMach[VECT_AX_TVL].xCMD	= VECT_Rst_OUT1; // TVL
						LED_Step = 0;

					}
					else if(!VectorStateMach[VECT_AX_TVL].xCmd_busy){

						VectorStateMach[VECT_AX_TVL].xCMD	= VECT_Rst_OUT1; // TVL
						_SR_Done = 1;
						LED_Indx++;
					}

				break;

				case 2:

					if(TML_MTR_INST[TML_AX_INDX].Error){

						VectorStateMach[VECT_AX_WF].xCMD	= VECT_Rst_OUT4; // OUT4 INDX
						LED_Step = 0;

					}
					else if(!VectorStateMach[VECT_AX_WF].xCmd_busy){

						VectorStateMach[VECT_AX_WF].xCMD	= VECT_Rst_OUT4; // OUT4 INDX
						_SR_Done = 1;
						LED_Indx++;
					}

				break;

				case 3:

					if(TML_MTR_INST[TML_AX_AHC].Error){

						VectorStateMach[VECT_AX_AHC].xCMD	= VECT_Rst_OUT0; // AHC
						LED_Step = 0;

					}
					else if(!VectorStateMach[VECT_AX_AHC].xCmd_busy){
						VectorStateMach[VECT_AX_AHC].xCMD	= VECT_Rst_OUT0; // AHC
						_SR_Done = 1;
						LED_Indx++;
					}

				break;

				case 4:

					if(TML_MTR_INST[TML_AX_OSC].Error){

						VectorStateMach[VECT_AX_OSC].xCMD	= VECT_Rst_OUT0; // OSC
						LED_Step = 0;

					}
					else if(!VectorStateMach[VECT_AX_OSC].xCmd_busy){
						VectorStateMach[VECT_AX_OSC].xCMD	= VECT_Rst_OUT0; // OSC
						_SR_Done = 1;
						LED_Indx++;
					}

				break;

				case 5:

					if(TML_MTR_INST[TML_AX_WF].Error){

						VectorStateMach[VECT_AX_WF].xCMD	= VECT_Rst_OUT1; // WF
						LED_Step = 0;

					}
					else if(!VectorStateMach[VECT_AX_WF].xCmd_busy){
						VectorStateMach[VECT_AX_WF].xCMD	= VECT_Rst_OUT1; // WF
						_SR_Done = 1;
						LED_Indx++;
					}

				break;

				case 6:

					if(TML_MTR_INST[TML_AX_INDX_EXT].Error){

						VectorStateMach[VECT_AX_TVL].xCMD	= VECT_Rst_OUT4; //
						LED_Step = 0;

					}
					else if(TML_MTR_INST[TML_AX_INDX_EXT].xCMD == TML_IDLE){
						VectorStateMach[VECT_AX_TVL].xCMD	= VECT_Rst_OUT4; //
						_SR_Done = 1;
						LED_Indx++;
					}

				break;

				default:

					LED_Indx = 0;

				break;
			}

			if(LED_Indx > 6){

				LED_Indx = 1;

			}

			if(_SR_Done){
				_SR_Done = 0;
				TimerStart(&LED_Tmr, KK_Blink);
				LED_Step = 41;

			}

		break;

		/////////////////////////////////////

		case 100:

			if(LED_CMD != 100){
				LED_Step = 0;
				LED_CMD = 0;
			}

			if(!TimerIsTimeOut(&LED_Tmr))
				break;

			if(LED_Indx == 0)
				LED_Indx = 1;

			switch(LED_Indx){

				case 1:

					if((!VectorStateMach[VECT_AX_TVL].xCmd_busy)
						|| (VectorStateMach[VECT_AX_TVL].xCMD >= VECT_Set_OUT0)){

						VectorStateMach[VECT_AX_TVL].xCMD 	= VECT_Set_OUT1; // TVL
						LED_Indx++;
					}

				break;

				case 2:

					if((!VectorStateMach[VECT_AX_WF].xCmd_busy)
						|| (VectorStateMach[VECT_AX_WF].xCMD >= VECT_Set_OUT0)){

						VectorStateMach[VECT_AX_WF].xCMD 	= VECT_Set_OUT4; // OUT4 INDX
						LED_Indx++;
					}

				break;

				case 3:

					if((!VectorStateMach[VECT_AX_AHC].xCmd_busy)
						|| (VectorStateMach[VECT_AX_AHC].xCMD >= VECT_Set_OUT0)){

						VectorStateMach[VECT_AX_AHC].xCMD 	= VECT_Set_OUT0; // AHC
						LED_Indx++;
					}

				break;

				case 4:

					if((!VectorStateMach[VECT_AX_OSC].xCmd_busy)
						|| (VectorStateMach[VECT_AX_OSC].xCMD >= VECT_Set_OUT0)){

						VectorStateMach[VECT_AX_OSC].xCMD 	= VECT_Set_OUT0; // OSC
						LED_Indx++;
					}

				break;

				case 5:

					if((!VectorStateMach[VECT_AX_WF].xCmd_busy)
						|| (VectorStateMach[VECT_AX_WF].xCMD >= VECT_Set_OUT1)){

						VectorStateMach[VECT_AX_WF].xCMD 	= VECT_Set_OUT0; // WF
						LED_Indx++;
					}

				break;

				case 6:

					if((!VectorStateMach[VECT_AX_TVL].xCmd_busy)
						|| (VectorStateMach[VECT_AX_TVL].xCMD >= VECT_Set_OUT4)){

						VectorStateMach[VECT_AX_TVL].xCMD 	= VECT_Set_OUT4; //
						LED_Indx++;
					}

				break;

				default:

					LED_Indx = 1;

					TimerStart(&LED_Tmr, 0.5);
					LED_Step = 101;

				break;
			}

		break;

		case 101:

			if(LED_CMD != 100){
				LED_Step = 0;
				LED_CMD = 0;
			}

			if(!TimerIsTimeOut(&LED_Tmr))
				break;

			if(LED_Indx == 0)
				LED_Indx = 1;

			switch(LED_Indx){

				case 1:

					if((!VectorStateMach[VECT_AX_TVL].xCmd_busy)
						|| (VectorStateMach[VECT_AX_TVL].xCMD >= VECT_Set_OUT0)){

						VectorStateMach[VECT_AX_TVL].xCMD 	= VECT_Rst_OUT1; // TVL
						LED_Indx++;
					}

				break;

				case 2:

					if((!VectorStateMach[VECT_AX_WF].xCmd_busy)
						|| (VectorStateMach[VECT_AX_WF].xCMD >= VECT_Set_OUT0)){

						VectorStateMach[VECT_AX_WF].xCMD 	= VECT_Rst_OUT4; // OUT4 INDX
						LED_Indx++;
					}

				break;

				case 3:

					if((!VectorStateMach[VECT_AX_AHC].xCmd_busy)
						|| (VectorStateMach[VECT_AX_AHC].xCMD >= VECT_Set_OUT0)){

						VectorStateMach[VECT_AX_AHC].xCMD 	= VECT_Rst_OUT0; // AHC
						LED_Indx++;
					}

				break;

				case 4:

					if((!VectorStateMach[VECT_AX_OSC].xCmd_busy)
						|| (VectorStateMach[VECT_AX_OSC].xCMD >= VECT_Set_OUT0)){

						VectorStateMach[VECT_AX_OSC].xCMD 	= VECT_Rst_OUT0; // OSC
						LED_Indx++;
					}

				break;

				case 5:

					if((!VectorStateMach[VECT_AX_WF].xCmd_busy)
						|| (VectorStateMach[VECT_AX_WF].xCMD >= VECT_Set_OUT1)){

						VectorStateMach[VECT_AX_WF].xCMD 	= VECT_Rst_OUT0; // WF
						LED_Indx++;
					}

				break;

				case 6:

					if((!VectorStateMach[VECT_AX_TVL].xCmd_busy)
						|| (VectorStateMach[VECT_AX_TVL].xCMD >= VECT_Set_OUT4)){

						VectorStateMach[VECT_AX_TVL].xCMD 	= VECT_Rst_OUT4; // EXT INDX
						LED_Indx++;
					}

				break;

				default:

					LED_Indx = 1;

					TimerStart(&LED_Tmr, 1.0);
					LED_Step = 100;

				break;
			}

		break;

	}

if(LED_Indx != _LED_Indx)
	LED_One_Blink_Req = 0;

_LED_Indx = LED_Indx;

return ;
}
```

### Program Logical/Tester (ANSIC)

#### Tester.c - Init, cyclic, exit code
```c
#include <bur/plctypes.h>

#ifdef _DEFAULT_INCLUDES
	#include <AsDefault.h>
#endif

_LOCAL INT MainCounter , CountPeriod , CountDelta , CountPeriod_SP;

INT _mainCounter;

INT Cntr_Incr(INT newVal , INT prevVal );

void _INIT ProgramInit(void)
{

  CountPeriod_SP =	2000;

}

void _CYCLIC ProgramCyclic(void)
{

	if(CountPeriod > CountPeriod_SP){
		CountPeriod = 0;

		CountDelta = Cntr_Incr(MainCounter , _mainCounter);

		_mainCounter = MainCounter;

	}
	else
		CountPeriod++;

	MainCounter--;
}

INT Cntr_Incr(INT newVal , INT prevVal ){
INT ret = 0;

	if(newVal < prevVal)
		return ((0xFFFF - prevVal)+ newVal + 1);
	else
		return (newVal - prevVal);

	return ret;
}
```

### Program Logical/HMI_Report (ANSIC)

#### HMI_Reports.c - Init, cyclic, exit code
```c
#include <bur/plctypes.h>

#ifdef _DEFAULT_INCLUDES
	#include <AsDefault.h>
#endif

//#include <..\Lib\statelib.c>
//#include <..\Lib\xstring.c>

#include <..\GlobalDef.h>
#include <..\GlobalDecl.h>

#include <..\Lib\Statelib.c>
#include <..\Lib\WSI_lib.c>
#include <..\Lib\LoggerLib.c>

#include<HMI_Reports.h>

_GLOBAL UINT Weld_Report_Status , Weld_Report_Start_Enable;

//////////////////////

_LOCAL UINT Page_Step;

_LOCAL DATE_AND_TIME LocalTime;

_LOCAL UINT KK_Catch;
_LOCAL UINT HMI_ClearError_vis;
_LOCAL plcbit HMI_ClearError_btn;

//_LOCAL plcstring KK_str[32] , KK_format[32];
//_LOCAL plcbit KK_CheckString;
//_LOCAL float KK_Float;
_LOCAL SINT KK_Result;
//_LOCAL USINT KK_dzien;

_LOCAL UINT HMI_Lock_Line[16] , HMI_Line_vis[16] , HMI_Ack_Btn_vis[16];
_LOCAL UINT NewFilePage_vis , _NewFilePage_vis , SetTimePage_vis , _SetTimePage_vis;
_LOCAL UINT HMI_Message_Vis;
_LOCAL UINT HMI_Head_Lock;
_LOCAL UINT Ack_Btn[16] , Glb_Ack_Btn , Glb_Ack_Btn_vis;
_LOCAL DTStructure HMI_DTStr;
_LOCAL DTStructure HMI_SetDTStr;
_LOCAL UINT HMI_Encoder_vis;
_LOCAL UINT HMI_InetrpassTemp_upd;
_LOCAL UINT HMI_HeatInput_vis[16] , HMI_PwrRatio_vis[16] , HMI_HeatInputLimit_vis , HMI_PwrRatioLimit_vis;
_LOCAL UINT HMI_UpdateLine;

_LOCAL float Freq , Dwell_In ,Dwell_Out;

//_LOCAL UDINT DwellIn_dec, DwellOut_dec , ExcurTime_dec;
//_LOCAL float _DwellIn, _DwellOut , _ExcurTime;

//  New File Name Data
_LOCAL plcstring HMI_File_BeadLog[16];
_LOCAL plcstring HMI_File_Name[64];
_LOCAL UINT HMI_File_LayerNo , HMI_File_BeadNo;
_LOCAL USINT HMI_File_TempEvery;
_LOCAL float HMI_File_WireDim;
_LOCAL double HMI_PowerRatio;
_LOCAL float HMI_HeatInput;
_LOCAL USINT HMI_PowerRatio_status;
_LOCAL UINT HMI_PowerRatio_Color;

/////////////////////////////
// new in July 2024

_LOCAL UINT HMI_Options_Vis;

///////
_LOCAL UINT GotoScreen , ReadPage , SetPage;

_LOCAL float _PowerRatio , KK_PowerRatio;
_LOCAL UINT LastBad_BEADS_Cnt;

_LOCAL DTSetTime_typ DTSetTime_1;

_LOCAL int _Len[8];

_LOCAL char LongBuf[512];
_LOCAL UDINT LongBufSize;

_LOCAL USINT TempEveryBead_Flag;

UINT _SeqStep;

void  MenuBar();
char* CreateHeaderTxt(char *p);

char* CreateLineTxt(char *p);

SINT IsItNumber(char*p);

float ActTemp();

void _INIT ProgramInit(void)
{
float f;

	//strcpy(KK_str , "80.2");

	strcpy(File_RW2.fileExten , ".txt");
	strcpy(File_RW2.deviceName, "REPORTS");

	//strcpy(KK_format ,"%2d");

	NewFilePage_vis = INVISIBLE;
	SetTimePage_vis = INVISIBLE;

	HMI_Message_Vis = INVISIBLE;

	HMI_Encoder_vis = INVISIBLE;

	HMI_Options_Vis = INVISIBLE;

	_SetTimePage_vis = SetTimePage_vis;

	HMI_PowerRatio_Color = 1;

	TempEveryBead_Flag = 1;

	if(ActTemp() > 340)
		Weld_Report_Status = 4; // Over temprature
	else
		Weld_Report_Status = 3; // Must enter temperature

	LastBad_BEADS_Cnt = Weld_Rep.BEADS_Cnt;

	/*

	if(CurCalib.GenFloatValue[SETUP_FLOAT_POWER_RATIO_LO] < 10.0)
		CurCalib.GenFloatValue[SETUP_FLOAT_POWER_RATIO_LO] = 10.0;

	if(CurCalib.GenFloatValue[SETUP_FLOAT_POWER_RATIO_HI] > 200.0)
		CurCalib.GenFloatValue[SETUP_FLOAT_POWER_RATIO_HI] = 200.0;

	*/

}

void _CYCLIC ProgramCyclic(void)
{
UINT i;
UINT status;
DTGetTime_typ dtGet;
float w1, w2 , f;

dtGet.enable = 1;
DTGetTime(&dtGet);
LocalTime = dtGet.DT1;

//Weld_Rep.Line[Weld_Rep.ActLINE].TimeStamp = dtGet.DT1;

/*

if(KK_CheckString){
	KK_CheckString = 0;

	KK_Result = IsItNumber(KK_str);
	xsprintf(KK_str , KK_format, KK_dzien);

}

if(OSC_TML_Param_Set[0].pDwell_In
	&& OSC_TML_Param_Set[0].pDwell_Out
	&& OSC_TML_Param_Set[0].pFreq){

	_DwellIn = (*OSC_TML_Param_Set[0].pDwell_In);
	_DwellOut = (*OSC_TML_Param_Set[0].pDwell_Out);
	_ExcurTime = (*OSC_TML_Param_Set[0].pFreq);

	DwellIn_dec = (UDINT)(_DwellIn * 10.0 +0.5);
	DwellOut_dec = (UDINT)(_DwellOut * 10.0 +0.5);
	ExcurTime_dec = (UDINT)(_ExcurTime * 10.0 +0.5);

}

*/

if((Weld_Rep.Report_Type == 0)){ // HEAT INPUT

		HMI_HeatInputLimit_vis = VISIBLE;
		HMI_PwrRatioLimit_vis = INVISIBLE;

	for(i = 0 ; i <16 ; i++){
		HMI_HeatInput_vis[i] =  HMI_Line_vis[i];
		HMI_PwrRatio_vis[i] = INVISIBLE;
	}

}
else{

		HMI_PwrRatioLimit_vis = VISIBLE;
		HMI_HeatInputLimit_vis = INVISIBLE;

	for(i = 0 ; i <16 ; i++){
			HMI_PwrRatio_vis[i] =	HMI_Line_vis[i];
			HMI_HeatInput_vis[i] = INVISIBLE;
		}
}

if((Weld_Report_Status < 2) // calculate only when begining and running
	|| HMI_UpdateLine
	|| HMI_InetrpassTemp_upd){ // or when line values are changed

	HMI_UpdateLine = 0;

	Weld_Rep.Line[Weld_Rep.ActLINE].TimeStamp = dtGet.DT1;

	/*

	if(PS_Param_Set[0].pAmpSP)
	  Weld_Rep.Line[Weld_Rep.ActLINE].PrimaryAmps = (*PS_Param_Set[0].pAmpSP);

	if(WIRE_Param_Set[0].pSpeedSp)
	  Weld_Rep.Line[Weld_Rep.ActLINE].PrimaryWireSpeed = (*WIRE_Param_Set[0].pSpeedSp) * 2.3622047244094488188976377952756;

	if(AVC_Param_Set[0].pVoltSP )
	  Weld_Rep.Line[Weld_Rep.ActLINE].PrimaryVolts = (*AVC_Param_Set[0].pVoltSP) ;

	if(OSC_TML_Param_Set[0].pFreq
		&& OSC_TML_Param_Set[0].pDwell_In
		&& OSC_TML_Param_Set[0].pDwell_Out){

		xsprintf(Weld_Rep.Line[Weld_Rep.ActLINE].Dwell_Excursion , "%d - %d - %d" , \
			(UDINT)((*OSC_TML_Param_Set[0].pDwell_In)*10.0 +0.5) , (UDINT)((*OSC_TML_Param_Set[0].pFreq)*10.0 +0.5) , (UDINT)((*OSC_TML_Param_Set[0].pDwell_Out)*10.0 +0.5));
	}

	*/

  	Weld_Rep.Line[Weld_Rep.ActLINE].PrimaryAmps = permMem.Analog_Out[AHCCurrentSPAO_Indx].Value;
  	Weld_Rep.Line[Weld_Rep.ActLINE].PrimaryWireSpeed = permMem.Analog_Out[WireFeedSpeedAO_Indx].Value; //  * 2.3622047244094488188976377952756;
  	Weld_Rep.Line[Weld_Rep.ActLINE].PrimaryVolts = permMem.Analog_Out[ArcVoltsAO_Indx].Value ;

	Freq = permMem.Analog_Out[OSCSpeedAO_Indx].Value;
	Dwell_In = permMem.Analog_Out[OSC_DwellInAO_Indx].Value;
	Dwell_Out = permMem.Analog_Out[OSC_DwellOutAO_Indx].Value;

	xsprintf(Weld_Rep.Line[Weld_Rep.ActLINE].Dwell_Excursion , "%d - %d - %d" , \
		(UDINT)(Dwell_In * 10.0 + 0.5) , (UDINT)( Freq * 10.0 + 0.5) , (UDINT)(Dwell_Out * 10.0 + 0.5));

	if(Weld_Rep.Line[Weld_Rep.ActLINE].Travel_Tungsten > 0.0){
		w1 =  Weld_Rep.Line[Weld_Rep.ActLINE].PrimaryAmps * Weld_Rep.Line[Weld_Rep.ActLINE].PrimaryVolts * 60.0;
			//Weld_Rep.Line[Weld_Rep.ActLINE].HeatInput = (w1/((*TVL_ROT_Param_Set[0].pPrimVel)* 2.3622047244094488188976377952756))*0.001;
		Weld_Rep.Line[Weld_Rep.ActLINE].HeatInput = (w1/Weld_Rep.Line[Weld_Rep.ActLINE].Travel_Tungsten)*0.001;
	}
	else
		Weld_Rep.Line[Weld_Rep.ActLINE].HeatInput = 0.0;

	HMI_HeatInput = Weld_Rep.Line[Weld_Rep.ActLINE].HeatInput;

	if(Weld_Rep.Line[Weld_Rep.ActLINE].Travel_Tungsten > 0.0){

		//w1 =  Weld_Rep.Line[Weld_Rep.ActLINE].PrimaryWireSpeed / (Weld_Rep.Line[Weld_Rep.ActLINE].Travel_Tungsten * 2.3622047244094488188976377952756);
		w1 =  Weld_Rep.Line[Weld_Rep.ActLINE].PrimaryWireSpeed / (Weld_Rep.Line[Weld_Rep.ActLINE].Travel_Tungsten);
		w2 = Weld_Rep.Head.WireDim/2.0;
		w2 = w2*w2 * M_PI;

		if((w1*w2) > 0){

			Weld_Rep.Line[Weld_Rep.ActLINE].PowerRatio = (Weld_Rep.Line[Weld_Rep.ActLINE].PrimaryVolts *Weld_Rep.Line[Weld_Rep.ActLINE].PrimaryAmps)/(w1 * w2)/1000.0;
		}
		else
			Weld_Rep.Line[Weld_Rep.ActLINE].PowerRatio = 0.0;

	}
	else
		Weld_Rep.Line[Weld_Rep.ActLINE].PowerRatio = 0.0;

	HMI_PowerRatio = Weld_Rep.Line[Weld_Rep.ActLINE].PowerRatio;

	//HMI_PowerRatio_status = ((HMI_PowerRatio >= 66.2) &&  (HMI_PowerRatio <= 87.6))? INVISIBLE:VISIBLE;

	Weld_Report_Start_Enable = 0;

	/*
	if((Weld_Rep.Report_Type == 0)){ // HEAT INPUT

		if(HMI_HeatInput < CurCalib.GenFloatValue[SETUP_FLOAT_HEAT_INPUT_LO])
			HMI_PowerRatio_Color = 84;

		else if(HMI_HeatInput > CurCalib.GenFloatValue[SETUP_FLOAT_HEAT_INPUT_HI])
			HMI_PowerRatio_Color = 43;

		else {

			HMI_PowerRatio_Color = 15;
			Weld_Report_Start_Enable = 1;

		}

	}else{

		if(HMI_PowerRatio < CurCalib.GenFloatValue[SETUP_FLOAT_POWER_RATIO_LO])
			HMI_PowerRatio_Color = 84;

		else if(HMI_PowerRatio > CurCalib.GenFloatValue[SETUP_FLOAT_POWER_RATIO_HI])
			HMI_PowerRatio_Color = 43;

		else {

			HMI_PowerRatio_Color = 15;
			Weld_Report_Start_Enable = 1;

		}

	}
	*/

	///* Test Radom
	/*
	if(Master[0].TestMode) // 11 Apr 2022
		Weld_Report_Start_Enable = 1;
	*/

}

else{

	/*
	if(Master[0].TestMode)  ///* Test Radom
		Weld_Report_Start_Enable = 1;
	else
		Weld_Report_Start_Enable = 0;
	*/

	HMI_PowerRatio_Color = 15;

}

/*
switch(CurCalib.GenSetup[SETUP_LOG_OPTION]){

	case 1: // Log After A side

		if(Weld_Report_Status == 2){ // Beat Finished

			if(Master[0].ToolHeadID){

				Weld_Report_Status = 0;
			}

		}

	break;

	case 2: // Log After B side

		if(Weld_Report_Status == 2){ // Beat Finished

			if(!Master[0].ToolHeadID){

				Weld_Report_Status = 0;
			}

		}

	break;

	case 3: // Log After Any Stop - // Allow beat log after any Stop

		if(!Master[0].SeqStep && _SeqStep)
			Weld_Report_Status = 2;

		if(Weld_Report_Status == 2)
			Weld_Report_Start_Enable = 1;

	break;

	default: break;

}

_SeqStep = Master[0].SeqStep;
*/

HMI_PowerRatio_status = (TempEveryBead_Flag > 0 )? VISIBLE:INVISIBLE;

/*

if(HMI_InetrpassTemp_upd){

	if(Weld_Report_Status == 3){ // Must enter temprature

		if(IsItNumber(Weld_Rep.Line[Weld_Rep.ActLINE].InetrpassTemp)>= 0){
			Weld_Report_Status = 0;
			TempEveryBead_Flag = 1;

		}

	}
}

*/

if(HMI_InetrpassTemp_upd){

	HMI_InetrpassTemp_upd = 0;

	if(IsItNumber(Weld_Rep.Line[Weld_Rep.ActLINE].InetrpassTemp)>= 0){

		f = ActTemp();

		if(f > 340.0 ){

			//if(Weld_Report_Status == 0)
				Weld_Report_Status = 4;

		}
		else if( (f < 320.0)  && ( f > 0.0)){

			if(Weld_Report_Status >= 3)
				Weld_Report_Status = 0; // over temperature - no Welding

		}

		if(Weld_Report_Status == 3){ // Must enter temprature

			Weld_Report_Status = 0;
			TempEveryBead_Flag = 1;

		}

		////////////////////

	}

}

if(Weld_Report_Status == 4)
	HMI_PowerRatio_Color = 87;

/////////////////////////
//////////////////

/////////////////////////////////////////////////////////
//Weld_Report_Mode = (CurCalib.GenSetup[SETUP_EXTRAS]&0x1)? 1:0;

//* Test Radom
if((Weld_Report_Status == 2)){
//if((Weld_Report_Status == 2) && !Master[0].TestMode){
 	HMI_Ack_Btn_vis[Weld_Rep.ActLINE] = VISIBLE;
	Glb_Ack_Btn_vis = VISIBLE;
}
else{

	HMI_Ack_Btn_vis[Weld_Rep.ActLINE] = INVISIBLE;
	Glb_Ack_Btn_vis = INVISIBLE;
}

if(NewFilePage_vis == VISIBLE){

	if(_NewFilePage_vis != NewFilePage_vis){

		strcpy(HMI_File_BeadLog , Weld_Rep.Head.WELD_LOG);
		HMI_File_LayerNo =   Weld_Rep.Head.LAYER_No;
		HMI_File_BeadNo = Weld_Rep.Line[0].BeadNo;
		HMI_File_TempEvery = Weld_Rep.Head.TempEvery;
		HMI_File_WireDim = Weld_Rep.Head.WireDim;

	}

	DT_TO_DTStructure(dtGet.DT1, (UDINT) &HMI_DTStr);
	xsprintf(HMI_File_Name, "%s-%d-%d %d-%d-%d %d-%d" , HMI_File_BeadLog , HMI_File_LayerNo , HMI_File_BeadNo , \
							HMI_DTStr.year , HMI_DTStr.month , HMI_DTStr.day , HMI_DTStr.hour , HMI_DTStr.minute);

}
_NewFilePage_vis = NewFilePage_vis;

if(SetTimePage_vis == VISIBLE){

	if(_SetTimePage_vis != SetTimePage_vis)
		DT_TO_DTStructure(LocalTime, (UDINT) &HMI_SetDTStr);

	if(DTSetTime_1.enable){

		DTSetTime_1.DT1 = DTStructure_TO_DT((UDINT) &HMI_SetDTStr);

		DTSetTime(&DTSetTime_1);
		if(!DTSetTime_1.status)
			DTSetTime_1.enable = 0;

		//SetTimePage_vis = INVISIBLE;

	}

}
_SetTimePage_vis = SetTimePage_vis;

////////////////
HMI_ClearError_vis = (File_RW2.Done && File_RW2.Error )? VISIBLE:INVISIBLE;

if(HMI_ClearError_btn){
	HMI_ClearError_btn = 0;

	File_RW2.Error = 0;
	File_RW2.Done = 0;
	File_RW2.CMD = 0;
	Page_Step = 0;

}
////////////////////

switch(Page_Step){

	default:

		GotoScreen = 10;

		if(Weld_Rep.ActLINE < 16 ){

			for (i = Weld_Rep.ActLINE ; i < 16 ; i++){

				HMI_Line_vis[i] = INVISIBLE;
				HMI_Ack_Btn_vis[i] = INVISIBLE;
			}

			for (i = 0 ; i < Weld_Rep.ActLINE ; i++){

					HMI_Line_vis[i] = VISIBLE;
					HMI_Ack_Btn_vis[i] = INVISIBLE;
					HMI_Lock_Line[i] = 1;
			}

		}
		else{

			Weld_Rep.ActLINE = 15;

			for (i = 0 ; i < 15 ; i++){

				HMI_Line_vis[i] = VISIBLE;
				HMI_Ack_Btn_vis[i] = INVISIBLE;
				HMI_Lock_Line[i] = 1;
			}

		}

		HMI_Lock_Line[Weld_Rep.ActLINE] = 0;
		HMI_Ack_Btn_vis[Weld_Rep.ActLINE] = VISIBLE;
		HMI_Line_vis[i] = VISIBLE;

		HMI_Head_Lock = (Weld_Rep.ActLINE > 0)? 1:0;

		HMI_Message_Vis = INVISIBLE;

		Page_Step = 1;

	break;

	case 1:	// Wait for Acknowledge Line

		status = 0;
		for(i = 0 ; i < 16 ; i++){

			if(Ack_Btn[i])
				status = i+1;

		}

		KK_Catch = status;

		if(status > 0 || Glb_Ack_Btn){

			Glb_Ack_Btn = 0;

			for(i = 0 ; i < 16 ; i++)
				Ack_Btn[i] = 0;

			Page_Step = 3;

		}

	break;

	case 3: // Add records TXT

		//NewFilePage_vis = INVISIBLE;

		KK_Result = IsItNumber(Weld_Rep.Line[Weld_Rep.ActLINE].InetrpassTemp);

		_PowerRatio = KK_PowerRatio;

		//status = ((_PowerRatio > 350) || (_PowerRatio < 340))? 1:0;
		//if(status)

		if(KK_Result >= 0){

			f = atof((UDINT) Weld_Rep.Line[Weld_Rep.ActLINE].InetrpassTemp);

			if(f > 340)
				TempEveryBead_Flag = 1;
			else if (f < 300)
				TempEveryBead_Flag = 0;

		}

		//if(HMI_PowerRatio_status == VISIBLE)
			//LastBad_BEADS_Cnt = Weld_Rep.BEADS_Cnt;

		if(TempEveryBead_Flag)
			LastBad_BEADS_Cnt = Weld_Rep.BEADS_Cnt;

		if(((KK_Result< 0))
			&& ((((Weld_Rep.BEADS_Cnt - LastBad_BEADS_Cnt)%(UINT)Weld_Rep.Head.TempEvery) == 0)
				|| (LastBad_BEADS_Cnt == Weld_Rep.BEADS_Cnt))){

			HMI_Message_Vis = VISIBLE;

			Page_Step = 1;

			break;
		}

		strcpy(File_RW2.fileName , Weld_Rep.FileName);
		strcat(File_RW2.fileName , File_RW2.fileExten);
		File_RW2.CMD = F_OPEN_ONLY;

		Page_Step ++;

	break;

	case 4:

		if(File_RW2.Done && !File_RW2.Error){

			if((File_RW2._int.FOpen.filelen == 0)){

				memset(&LongBuf[0] , 0 , 512);
				LongBufSize = 0;

				Weld_Rep.BEADS_Cnt = 1;

				//CreateHeaderTxt(&LongBuf[0]);
				CreateLineTxt(CreateHeaderTxt(LongBuf));

				//File_RW2.pMem = LongBuf;
				//File_RW2.Len = LongBufSize;
				//File_RW2.Offset = 0;

			}
			else{

				for(i = 0 ; i < 512 ; i++)
					LongBuf[i] = 0;

				//memset(&LongBuf[0] , 0 , 512);
				LongBufSize = 0;

				Weld_Rep.BEADS_Cnt++;

				CreateLineTxt(LongBuf);

			}

			File_RW2.pMem = LongBuf;
			File_RW2.Len = LongBufSize;
			File_RW2.Offset = File_RW2._int.FOpen.filelen;

			HMI_Head_Lock = 1;
			File_RW2.CMD = F_WRITE_ONLY;

			Page_Step ++;

		}
		else if(File_RW2.Error){

			//Page_Step = 0;
		}

	break;

	case 5:

		if(File_RW2.Done && !File_RW2.Error ){

			File_RW2.CMD = F_CLOSE_ONLY;

			Page_Step ++;

		}
		else if(File_RW2.Error){

			//Page_Step = 0;
		}

	break;

	case 6:

		if(File_RW2.Done){

			if(File_RW2.Error){

				//Page_Step = 0;

			}else{

				if(Weld_Rep.ActLINE < 15 ){

					HMI_Lock_Line[Weld_Rep.ActLINE] = 1;
					HMI_Ack_Btn_vis[Weld_Rep.ActLINE] = INVISIBLE;
					Weld_Rep.ActLINE++;
					HMI_Line_vis[Weld_Rep.ActLINE] = VISIBLE;
					HMI_Lock_Line[Weld_Rep.ActLINE] = 0;
					HMI_Ack_Btn_vis[Weld_Rep.ActLINE] = VISIBLE;

					i = Weld_Rep.ActLINE;

					memcpy(&Weld_Rep.Line[i] , &Weld_Rep.Line[i-1] , sizeof(Weld_Report_Line_typ));

				}else{

					for(i = 1 ; i < 16 ; i++)
						memcpy(&Weld_Rep.Line[i-1] , &Weld_Rep.Line[i] , sizeof(Weld_Report_Line_typ));

					i = 15;
				}

				Weld_Rep.Line[i].BeadNo = Weld_Rep.Line[i-1].BeadNo + 1;

				if(ActTemp() < 340.0)
				 	strcpy(Weld_Rep.Line[i].InetrpassTemp , "");

				strcpy(Weld_Rep.Line[i].Comments , "");

				if(ActTemp() > 340)
					Weld_Report_Status = 4;
				else
					Weld_Report_Status = 0;

				Page_Step = 1;

			}

		}

	break;

	//////////////////    New Report TXT ////////////////////////////
	 case 80:

		strcpy(Weld_Rep.Head.WELD_LOG , HMI_File_BeadLog);
		Weld_Rep.Head.LAYER_No = HMI_File_LayerNo;
		Weld_Rep.Line[0].BeadNo = HMI_File_BeadNo;
		Weld_Rep.Head.TempEvery = HMI_File_TempEvery;
		Weld_Rep.Head.WireDim = HMI_File_WireDim;
		//'%0.2d'
		DT_TO_DTStructure(dtGet.DT1, (UDINT) &HMI_DTStr);
		xsprintf(Weld_Rep.FileName, "%s-%d-%d %d-%0.2d-%0.2d %0.2d-%0.2d" , Weld_Rep.Head.WELD_LOG , Weld_Rep.Head.LAYER_No , Weld_Rep.Line[0].BeadNo , \
											HMI_DTStr.year , HMI_DTStr.month , HMI_DTStr.day , HMI_DTStr.hour , HMI_DTStr.minute);

		if(Weld_Rep.Head.WireDim <= 0.0)
			Weld_Rep.Head.WireDim = 0.045;

		if(Weld_Rep.Head.TempEvery == 0)
			Weld_Rep.Head.TempEvery = 4;

		i = 0;

		xsprintf(Weld_Rep.Line[i].WelderStamp,"RB 22%d", (DINT)i+1);

		Weld_Rep.Line[i].PrimaryAmps = 100.0;
		Weld_Rep.Line[i].PrimaryWireSpeed = 200.0;
		Weld_Rep.Line[i].PrimaryVolts = 10.0;
		Weld_Rep.Line[i].Travel_Tungsten = 3.0;
		Weld_Rep.Line[i].PowerRatio = 75.0;
		strcpy(Weld_Rep.Line[i].InetrpassTemp , "");
		xsprintf(Weld_Rep.Line[i].Dwell_Excursion,"%d - %d - %d", (i%10) , ((i+1)%10) , ((i+2)%10));

		xsprintf(Weld_Rep.Line[i].Comments,"");

		Weld_Rep.BEADS_Cnt = 0;
		Weld_Rep.LINES_Offset = 0;
		Weld_Rep.ActLINE = 0;

		HMI_Line_vis[0] = VISIBLE;
		HMI_Ack_Btn_vis[0] = VISIBLE;
		HMI_Lock_Line[0] = 0;

		HMI_Head_Lock = 0;

		for (i = 1 ; i < 16 ; i++){

			HMI_Line_vis[i] = INVISIBLE;
			HMI_Ack_Btn_vis[i] = INVISIBLE;
		}

		Page_Step ++;

	 break;

	 case 81:

	 	strcpy(File_RW2.fileNewName , Weld_Rep.FileName);
		File_RW2.CMD = F_WRITE;
	 	File_RW2.pMem =&Weld_Rep;
		File_RW2.Len = 0;
		File_RW2.Offset = 0;;

		Page_Step ++;

	 break;

	 case 82:

	 	if(File_RW2.Done){

			if(File_RW2.Error){

				//Page_Step = 0;
			}
			else{

				NewFilePage_vis = INVISIBLE;
				Page_Step = 1;

				Weld_Report_Status = 3;
				LastBad_BEADS_Cnt = Weld_Rep.BEADS_Cnt;
			}

	 	}

	 break;

}

MenuBar();
/////////////////////////////////////////////////////////

	/**************************************************/
	pFileRW = (FILE2_RW_typ*) &File_RW2;

	/*************************************************/
	if((pFileRW->CMD == 0)){

		pFileRW->Tmr.IN = 0;
		pFileRW->Tmr.Q = 0;

	}

	else if(TimerIsTimeOut(&pFileRW->Tmr)){

		pFileRW->Tmr.IN = 0;
		pFileRW->Tmr.Q = 0;

	}
	/**********************************************/

	if(pFileRW->_int.step == 0){

		if(pFileRW->CMD && !_CMD){

			switch(pFileRW->CMD){

				default:
					TimerStart(&pFileRW->Tmr, 10.0); // 15 sec to run command
				break;
			}

		}

		switch(pFileRW->CMD){

			case F_WRITE:

				//strcpy(pFileRW->fileNewName , pFileRW->fileNewName);

				DeleteExtension(pFileRW->fileNewName);
				strcat(pFileRW->fileNewName , pFileRW->fileExten);

				pFileRW->Error = 0;
				strcpy(pFileRW->MsgText , "");
				pFileRW->Done  = 0;
				pFileRW->_int.step = 50;

			break;

			case F_OPEN_ONLY:

				pFileRW->Error = 0;
				strcpy(pFileRW->MsgText , "");
				pFileRW->Done  = 0;
				pFileRW->_int.step = 120;

			break;

			case F_WRITE_ONLY:

				pFileRW->Error = 0;
				strcpy(pFileRW->MsgText , "");
				pFileRW->Done  = 0;
				pFileRW->_int.step = 140;

			break;

			case F_CLOSE_ONLY:

				pFileRW->Error = 0;
				strcpy(pFileRW->MsgText , "");
				pFileRW->Done  = 0;
				pFileRW->_int.step = 150;

			break;

			default:

				if(pFileRW->CMD)
					pFileRW->_int.step = 254;  // error

			break;

		 }

		/////////////////////////////////
		_CMD = pFileRW->CMD;

	}
	/********************************************/

	switch (pFileRW->_int.step )
  	{

		case 0: /**** First step ****/

			pFileRW->CMD = 0;

		break;

		////////    //////////////////////

		case 50: /**** open existing file ****/

			strcpy(pFileRW->fileName ,pFileRW->fileNewName );

			_Open(pFileRW);

			 if (pFileRW->_int.wStatus == ERR_OK)
			{

					pFileRW->_int.step ++;

			}
			else if (pFileRW->_int.wStatus == fiERR_FILE_NOT_FOUND )
			{

				pFileRW->_int.step += 2;

			}
			else if (pFileRW->_int.wStatus != 65535)
			{
				pFileRW->_int.byErrorLevel = 1;
				pFileRW->_int.step  = 254; // Error

			if (pFileRW->_int.wStatus == 20799)
			{
			  pFileRW->_int.wError = FileIoGetSysError();
			}
			}
		break;

		case 51: /**** Delete file ****/

			_Delete(pFileRW);

			/* Verify status */
			/* Verify status */
			if (pFileRW->_int.wStatus == 0)		   {

		   	 	pFileRW->_int.step ++;
		   }

		   else if (pFileRW->_int.wStatus != 65535)
		   {
			  pFileRW->_int.byErrorLevel = 7;
			  pFileRW->_int.step  = 254; // Error

			  if (pFileRW->_int.wStatus == 20799)
			  {
				 pFileRW->_int.wError = FileIoGetSysError();
			  }
			}
		break;

		case 52: /**** Create file ****/

			_Create(pFileRW);

			/* Verify status */
			if (pFileRW->_int.wStatus == 0)
			{

			 	pFileRW->_int.step++;
			}
			else if (pFileRW->_int.wStatus != 65535)
			{
				pFileRW->_int.byErrorLevel = 2;
				pFileRW->_int.step  = 254; // Error

				if (pFileRW->_int.wStatus == 20799)
				{
					pFileRW->_int.wError = FileIoGetSysError();
				}
			}

		break;

		case 53: /**** Write data ****/

			_Write(pFileRW);

			if (pFileRW->_int.wStatus == 0)
			{

			  	pFileRW->_int.step++;

			}
			else if (pFileRW->_int.wStatus != 65535)
			{
				pFileRW->_int.byErrorLevel = 6;
			  	pFileRW->_int.step  = 254; // Error

				if (pFileRW->_int.wStatus == 20799)
				{
				 	pFileRW->_int.wError = FileIoGetSysError();
				}
			}

		break;

		case 54: /**** Close file ****/

			_Close(pFileRW);

			//pFileRW->_int.PathDoneCnt = 0;

		   if (pFileRW->_int.wStatus == 0)
		   {

				DeleteExtension(pFileRW->fileName);

				//pFileRW->_int.step = 62; // get new directory info into string

				pFileRW->_int.step  = 255; // Success

		   }
		   else if (pFileRW->_int.wStatus != 65535)
		   {
			  pFileRW->_int.byErrorLevel = 5;
			  pFileRW->_int.step  = 254; // Error

			  if (pFileRW->_int.wStatus == 20799)
			  {
				 pFileRW->_int.wError = FileIoGetSysError();
			  }
			}
		break;

		//////////////////////////////////////////////////////

		case 120: /** OPEN ONLY **/

			_Open(pFileRW);

			/* Verify status */
			if (pFileRW->_int.wStatus == 0)
			{
				 pFileRW->_int.step  = 255; // Success
			}
			else if (pFileRW->_int.wStatus != 65535)
			{
				pFileRW->_int.byErrorLevel = 4;

				pFileRW->_int.step  = 254; // Error

				if (pFileRW->_int.wStatus == 20799)
					pFileRW->_int.wError = FileIoGetSysError();

			}

		break;

		//////////////////////////////////////////////////////

		case 140: /** Write ONLY **/

			_Write(pFileRW);

			/* Verify status */
			if (pFileRW->_int.wStatus == 0)
			{
				 pFileRW->_int.step  = 255; // Success
			}
			else if (pFileRW->_int.wStatus != 65535)
			{
				pFileRW->_int.byErrorLevel = 4;

				pFileRW->_int.step  = 254; // Error

				if (pFileRW->_int.wStatus == 20799)
					pFileRW->_int.wError = FileIoGetSysError();

			}

		break;

		//////////////////////////////////////////////////////

		case 150: /** Close ONLY **/

			_Close(pFileRW);

			/* Verify status */
			if (pFileRW->_int.wStatus == 0)
			{
				 pFileRW->_int.step  = 255; // Success
			}
			else if (pFileRW->_int.wStatus != 65535)
			{
				pFileRW->_int.byErrorLevel = 4;

				pFileRW->_int.step	= 254; // Error

				if (pFileRW->_int.wStatus == 20799)
					pFileRW->_int.wError = FileIoGetSysError();

			}

		break;

		////////////////////////////////////////////////////////
		// Error

		case 254: /**** Error ****/

			switch(pFileRW->_int.wStatus){

				case 9999: //ERR_NOTIMPLEMENTED
					strcpy(pFileRW->MsgText , "Err: not Implemented"); break;

				case 20700: //fiERR_INVALID_PATH
					strcpy(pFileRW->MsgText , "Err: Invalid Path"); break;

				case 20705: //fiERR_EXIST
					strcpy(pFileRW->MsgText , "Err: File Already Exist"); break;

				case 20799: //fiERR_SYSTEM
					strcpy(pFileRW->MsgText , "Err: System "); break;

				case 20798://fiERR_DEVICE_MANAGER
					strcpy(pFileRW->MsgText , "Err: Device Manager"); break;

				case 20797: //fiERR_DEVICE_DRIVER
					strcpy(pFileRW->MsgText , "Err: Device Driver"); break;

				case 20725: //fiERR_DIR_ALREADY_EXIST
					strcpy(pFileRW->MsgText , "Err: Directory Already Exist"); break;

				case 20724: //fiERR_DIR_NOT_EMPTY
					strcpy(pFileRW->MsgText , "Err: Directory Not Empty"); break;

				case 20723: //fiERR_DIR_NOT_EXIST
					strcpy(pFileRW->MsgText , "Err: Directory Not Exist"); break;

				case 20722: //fiERR_INVALID_DIRECTORY
					strcpy(pFileRW->MsgText , "Err: Invalid Directory"); break;

				case 20721:	//fiERR_FILE_NOT_OPENED
					strcpy(pFileRW->MsgText , "Err: File Not Opened"); break;

				case 20718:	//fiERR_COM_FILE_IOCTL
					strcpy(pFileRW->MsgText , "Err: File IO Control"); break;

				case 20717: //fiERR_COM_FILE_WRITE
					strcpy(pFileRW->MsgText , "Err: File Write"); break;

				case 20716:	//fiERR_COM_FILE_READ
					strcpy(pFileRW->MsgText , "Err: File Read"); break;

				case 20715:	//fiERR_COM_FILE_CLOSE
					strcpy(pFileRW->MsgText , "Err: File Close"); break;

				case 20714:	//fiERR_COM_FILE_OPEN
					strcpy(pFileRW->MsgText , "Err: File Open"); break;

				case 20708:	//fiERR_FILE_NOT_FOUND
					strcpy( pFileRW->MsgText , "Err: File Not Found"); break;

				default: strcpy( pFileRW->MsgText , "Err: Unknown"); break;
				//default: xsprintf(pFileRW->MsgText , "Err.Cmd: %d Code %d" , pFileRW->CMD , pFileRW->_int.wStatus); break;

			}

			PleaseShowFileMessage = 1;

			DeleteExtension(pFileRW->fileName);
			DeleteExtension(pFileRW->fileNewName);

			pFileRW->Error = 1;
			pFileRW->Done  = 1;
			pFileRW->_int.step  = 0;
			pFileRW->CMD = 0;

		break;

		case 255: /**** Success****/

			DeleteExtension(pFileRW->fileName);
			DeleteExtension(pFileRW->fileNewName);

			pFileRW->Error = 0;
			pFileRW->Done  = 1;
			pFileRW->_int.step  = 0;

			switch(	pFileRW->CMD){

				case F_READ: 				strcpy(pFileRW->MsgText , "F_READ Done" ); PleaseShowFileMessage = 1; break;
				case F_WRITE: 				strcpy(pFileRW->MsgText , "F_WRITE Done");  PleaseShowFileMessage = 1; break;
				case F_DELETE: 				strcpy(pFileRW->MsgText , "F_DELETE Done");  PleaseShowFileMessage = 1; break;
				case F_FREE_MEM: 			strcpy(pFileRW->MsgText , "F_FREE_MEM"); break;

				case F_RENAME: 				strcpy(pFileRW->MsgText , "F_RENAME Done" );  PleaseShowFileMessage = 1; break;
				case F_COPY: 				strcpy(pFileRW->MsgText , "F_COPY Done" );  PleaseShowFileMessage = 1; break;

				//case F_READ_FILE_TO_TMP: 	strcpy(pFileRW->MsgText , "F_READ_FILE_TO_TMP"); break;
				//case F_SAVE_AS_TMP: 		strcpy(pFileRW->MsgText , "F_SAVE_AS_TMP"); break;

				case F_READ_DIR: 			strcpy(pFileRW->MsgText , "F_READ_DIR"); break;
				case F_READ_FILE_INF: 		strcpy(pFileRW->MsgText , "F_READ_FILE_INF"); break;
				case F_READ_DIR_FILELIST: 	strcpy(pFileRW->MsgText , "F_READ_DIR_FILELIST"); break;

			}

			pFileRW->CMD = 0;

		break;

  }
	TimerExecute(&pFileRW->Tmr);
}

void _Open(FILE2_RW_typ *f)
{

	f->_int.FOpen.enable		= 1;
	f->_int.FOpen.pDevice   = (UDINT)f->deviceName;
	f->_int.FOpen.pFile = (UDINT)f->fileName;
	f->_int.FOpen.mode	  = FILE_RW;
	FileOpen(&f->_int.FOpen);

	f->_int.dwIdent = f->_int.FOpen.ident;
	f->_int.wStatus = f->_int.FOpen.status;

	return;
}
void _Close(FILE2_RW_typ *f){

	f->_int.FClose.enable	 = 1;
	f->_int.FClose.ident 	 = f->_int.dwIdent;
	FileClose(&f->_int.FClose);

	f->_int.wStatus = f->_int.FClose.status;

	return;

}
void _Create(FILE2_RW_typ *f){

	f->_int.FCreate.enable	= 1;
	f->_int.FCreate.pDevice = (UDINT) f->deviceName;
	f->_int.FCreate.pFile   = (UDINT)f->fileNewName;
	FileCreate(&f->_int.FCreate);

	f->_int.dwIdent = f->_int.FCreate.ident;
	f->_int.wStatus = f->_int.FCreate.status;

	return;

}

void _Write(FILE2_RW_typ *f){

	f->_int.FWrite.enable   = 1;
	f->_int.FWrite.ident    = f->_int.dwIdent;
	f->_int.FWrite.offset   = f->Offset;
	f->_int.FWrite.pSrc	   = f->pMem;
	f->_int.FWrite.len	   = f->Len;

	FileWrite(&f->_int.FWrite);

	f->_int.wStatus = f->_int.FWrite.status;

	return;

}

void _Delete(FILE2_RW_typ *f){

	f->_int.FDelete.enable	 = 1;
	f->_int.FDelete.pDevice = (UDINT) f->deviceName;
	f->_int.FDelete.pName	=  (UDINT)f->fileName;
	/* Call FBK */
	FileDelete(&f->_int.FDelete);
	/* Get status */
	f->_int.wStatus = f->_int.FDelete.status;

	return;
}

void DeleteExtension(char *p){

UINT len , i;

	len = strlen(p);

	for(i=0 ; i < len ; i++){

		if(p[i]=='.'){

			p[i] = 0;
			break;

		}

	}

	return;

}

void  MenuBar(){

	if ( GotoScreen < 0xFFFF ) {

		if(GotoScreen >= 10){
			if(GotoScreen != ReadPage) {

				//Screen.ReturnScreen	= Screen.ReadPage;
				SetPage = GotoScreen;

			}
			GotoScreen 	= 0xFFFF;
		}
	}

return;
}

char* CreateHeaderTxt(char *p){

	xsprintf(p ,"\t WELD OPERATOR BEAD LOG - \t %s \n\n WELD No.:\t %s \t" ,\
		Weld_Rep.Head.WELD_LOG , Weld_Rep.Head.WELD_No);

	_Len[0] = strlen(p); p+=_Len[0];

	xsprintf(p ,"\t WIRE HEAT No.: \t %s \t \tMACHINE I.D.: \t %s \n\n" , \
		Weld_Rep.Head.WIRE_HEAT_No , Weld_Rep.Head.MACHINE_Id);
	_Len[1] = strlen(p); p+=_Len[1];

	xsprintf(p ,"LAYER No.:\t %d \t\t WPS:\t %s \t\tM_TE:\t %s \t\t Cal.Due:\t %s \n\n"\
			, Weld_Rep.Head.LAYER_No , Weld_Rep.Head.WPS , Weld_Rep.Head.M_TE , Weld_Rep.Head.Cal_Due );
	_Len[2] = strlen(p); p+=_Len[2];

	xsprintf(p ,"Welder\t \tBead\t Primary\t Primary\t Primary\t Dwell Out / \t");
	_Len[3] = strlen(p); p+=_Len[3];

	//xsprintf(p ,"Travel @\tPower Ratio)\t Interpass\t \n");
	//xsprintf(p ,"Travel @\tPower Ratio)\t Heat Input\t Interpass\t \n");
	xsprintf(p ,"Travel @\tPower Ratio)\t Interpass\t \n");
	_Len[4] = strlen(p); p+=_Len[4];

	xsprintf(p ,"Stamp No.\t Date\tNo. \t Amps\t Wire Speed \t Volts \tExcur/Dwell In\t");
	_Len[5] = strlen(p); p+=_Len[5];

	//xsprintf(p ,"Tungsten\t (kW/in2)\t (kJ)\t Temp (F)\t Comments \n");
	xsprintf(p ,"Tungsten\t (kW/in2)\t Temp (F)\t Comments \n");
	_Len[6] = strlen(p); p+=_Len[6];

	LongBufSize += _Len[0] + _Len[1] + _Len[2] + _Len[3] + _Len[4] + _Len[5] + _Len[6];

	return p;

}

char* CreateLineTxt(char *p){
DTStructure DTStr;

	if(Weld_Rep.ActLINE >= 16)
		Weld_Rep.ActLINE = 15;

	DT_TO_DTStructure(Weld_Rep.Line[Weld_Rep.ActLINE].TimeStamp, (UDINT) &DTStr);

	//xsprintf(p ,"%s\t %d/%d/%d %d:%d \t" ,
	xsprintf(p ,"%s\t %0.2d/%0.2d/%d %0.2d:%0.2d:%0.2d \t" ,\
		Weld_Rep.Line[Weld_Rep.ActLINE].WelderStamp , DTStr.month ,  DTStr.day ,   DTStr.year , DTStr.hour , DTStr.minute , DTStr.second);
	_Len[0] = strlen(p); p+=_Len[0];

/*
	xsprintf(p ," %d \t %f \t %f \t %4.1f \t %s \t %4.1f \t %4.1f \t %4.1f \t %s \t %s \t \n" ,
			Weld_Rep.Line[Weld_Rep.ActLINE].BeadNo , Weld_Rep.Line[Weld_Rep.ActLINE].PrimaryAmps , Weld_Rep.Line[Weld_Rep.ActLINE].PrimaryWireSpeed , \
			Weld_Rep.Line[Weld_Rep.ActLINE].PrimaryVolts , Weld_Rep.Line[Weld_Rep.ActLINE].Dwell_Excursion , Weld_Rep.Line[Weld_Rep.ActLINE].Travel_Tungsten ,\
			Weld_Rep.Line[Weld_Rep.ActLINE].PowerRatio , Weld_Rep.Line[Weld_Rep.ActLINE].HeatInput , Weld_Rep.Line[Weld_Rep.ActLINE].InetrpassTemp , Weld_Rep.Line[Weld_Rep.ActLINE].Comments );
*/

	xsprintf(p ," %d \t %f \t %f \t %4.1f \t %s \t %4.1f \t %4.1f \t %s \t %s \t \n" ,
			Weld_Rep.Line[Weld_Rep.ActLINE].BeadNo , Weld_Rep.Line[Weld_Rep.ActLINE].PrimaryAmps , Weld_Rep.Line[Weld_Rep.ActLINE].PrimaryWireSpeed , \
			Weld_Rep.Line[Weld_Rep.ActLINE].PrimaryVolts , Weld_Rep.Line[Weld_Rep.ActLINE].Dwell_Excursion , Weld_Rep.Line[Weld_Rep.ActLINE].Travel_Tungsten ,\
			Weld_Rep.Line[Weld_Rep.ActLINE].PowerRatio  , Weld_Rep.Line[Weld_Rep.ActLINE].InetrpassTemp , Weld_Rep.Line[Weld_Rep.ActLINE].Comments );

	_Len[1] = strlen(p); p+=_Len[1];

	LongBufSize += _Len[0] + _Len[1];

	return p;
}

SINT IsItNumber(char*p){
UINT len;
SINT status;

	len = 0;
	status = 0;

	while((*p!= 0) && (len < 10) && (status >= 0)){

		if(*p == '.'){

			if(status == 0)
				status = 1;
			else
				status = -1;

		}
		else if((*p < '0') || (*p > '9'))
			status = -2;

		p++;
		len++;

	}

	if(len == 0)
		status = -3;

	return status;

}

float ActTemp(){

float ret;

	if(IsItNumber(Weld_Rep.Line[Weld_Rep.ActLINE].InetrpassTemp)>= 0){

		ret = atof((UDINT) Weld_Rep.Line[Weld_Rep.ActLINE].InetrpassTemp);

	}
	else
		ret = 0.0;

	return ret;

}
```

#### HMI_Reports.h
```c
#include <math.h>

/*

#include <..\GlobDef.h>
#include <..\..\Lib\WSI_Lib.c>

#include <..\GlobDecl.h>
#include <..\Hardcoded.c>
#include <..\HMI_Cntrl.c>
#include <..\HeadConfig.c>

#include <..\..\Lib\Statelib.c>
#include <..\..\Lib\LCDLib.c>
#include <..\..\Lib\LoggerLib.c>
*/

#ifndef _HMI_REPORTS_
#define _HMI_REPORTS_

/*********************************************************************/
typedef struct FILEIO2_RW_HS_INT_typ
{
	UINT 		   step;
	USINT          byErrorLevel;
	UINT           wStatus;
	UINT           wError;
	UDINT          dwIdent;
	UDINT 		   memlng;

	FileOpen_typ   FOpen;
	FileClose_typ  FClose;
	FileCreate_typ FCreate;
	FileRead_typ   FRead;
	FileWrite_typ  FWrite;
	FileDelete_typ FDelete;
	DirInfo_typ	   FDirInfo;
	DirRead_typ	   FFileInfo;

	FileRename_typ FRename;
	FileCopy_typ   FCopy;

	//UDINT OffsetToWeldProgramLinkMode;
	//UDINT OffsetToWeldProgramRepeat;

	//UINT  PathDoneCnt;

}FILEIO2_RW_HS_INT_typ;

typedef struct FILE2_RW_typ
{

	USINT CMD;
	plcbit Done;
	plcbit Error;
	plcbit FileLocked;
	plcbit NewFileLoaded;
	USINT Mode;

	plcstring fileName[64];
	plcstring fileNewName[64];
	plcstring fileExten[6];

	plcstring deviceName[32];
	plcstring targetDeviceName[32];

	UINT TargetDevice_Indx;
	UINT SourceDevice_Indx;

	UINT DirList_Page[2];

	plcstring MsgText[128];
	UDINT FilesNum[2];
	UINT DirList_Page_Num[2];

	fiDIR_READ_DATA  FileInfo[1];

	TON_typ Tmr;

	UDINT pMem;
	UDINT Len;
	UDINT Offset;

	FILEIO2_RW_HS_INT_typ _int;

}FILE2_RW_typ;

/***********************************************/
typedef struct Weld_Report_Line_typ
{
	plcstring WelderStamp[16];
	DATE_AND_TIME TimeStamp;
	UINT BeadNo;
	float PrimaryAmps;
	float PrimaryWireSpeed;
	float PrimaryVolts;
	plcstring  Dwell_Excursion[16];
	float Travel_Tungsten;
	float PowerRatio;
	float HeatInput;
	plcstring InetrpassTemp[8];
	plcstring  Comments[32];

}Weld_Report_Line_typ;

typedef struct Weld_Report_Head_typ
{
plcstring WELD_LOG[16];
plcstring WELD_No[16];
plcstring WIRE_HEAT_No[16];
plcstring MACHINE_Id[16];
UINT LAYER_No;
plcstring WPS[16];
plcstring M_TE[16];
plcstring Cal_Due[16];
float WireDim;
USINT TempEvery;

}Weld_Report_Head_typ;

typedef struct Weld_Report_typ
{
plcstring FileName[64];
UINT LINES_No;
UINT LINES_Offset;
UINT ActLINE;
UINT BEADS_Cnt;
UINT Report_Type;
Weld_Report_Head_typ Head;
Weld_Report_Line_typ Line[16];

}Weld_Report_typ;

/*
typedef struct Weld_Report_Line_typ
{
	plcstring delimit_begin[4];
	plcstring WelderStamp[16];
	plcstring delimit_1[4];
	plcstring TimeStamp[16];
	plcstring delimit_2[4];
	plcstring BeadNo[8];
	plcstring delimit_3[4];
	plcstring PrimaryAmps[8];
	plcstring PrimaryWireSpeed[8];
	plcstring PrimaryVolts[8];
	plcstring Dwell_Excursion[16];
	plcstring Travel_Tungsten;
	float PowerRatio;
	float InetrpassTemp;
	plcstring  Comments[32];

}Weld_Report_Line_typ;

*/

/***********************************************/

/********			 Files Operetion	    **********/

/***********************************************/

#define PRG_FILE_EXT ".prg"
#define PRG_NO_NEXT "None"

#define F_READ 				1
#define F_WRITE 			2
#define F_DELETE			3
#define F_FREE_MEM 			4

#define F_RENAME			8
#define F_COPY				9

#define F_READ_DIR 			20
#define F_READ_FILE_INF 	21
#define F_READ_DIR_FILELIST 22

#define F_OPEN_ONLY 		30
#define F_CREATE_ONLY 		31
#define F_WRITE_ONLY 		32
#define F_CLOSE_ONLY 		33
#define F_READ_ONLY 		34

/*

#define F_READ 				1
#define F_WRITE 			2
#define F_DELETE			3
#define F_FREE_MEM 			4

#define F_LOAD_CURCFG		5
#define F_SAVE_CURCFG		6
#define F_SAVE_AS_CURCFG	7

#define F_RENAME			8
#define F_COPY				9
#define F_GET_NEXT_FILE		10
#define F_SET_NEXT_FILE		11
#define F_READ_FILE_TO_TMP 	12
#define F_SAVE_AS_TMP 		13

#define F_READ_DIR 			20
#define F_READ_FILE_INF 	21
#define F_READ_DIR_FILELIST 22

#define F_OPEN_ONLY 		30
#define F_CREATE_ONLY 		31
#define F_WRITE_ONLY 		32
#define F_CLOSE_ONLY 		33

#define F_READ_FILES_CHAIN  40
#define F_EDIT_CHAIN  		41

#define F_SAVE_CURCFG_BIN		45
#define F_SAVE_AS_CURCFG_BIN	46
#define F_SAVE_SETUP_BIN		47
#define F_SAVE_AS_FULL_BIN		48
#define F_SAVE_AS_CALIB_BIN		49

#define F_MODE_BINARY		0
#define F_MODE_XML			1
#define F_MODE_BINARY_FULL	2
#define F_MODE_BINARY_CALIB	3

*/

#define CF_DEV_INDX 0
#define	USB_DEV_INDX 1

#define VISIBLE 	0
#define INVISIBLE 	1
/******************************************************/
_GLOBAL_RETAIN Weld_Report_typ Weld_Rep;

_GLOBAL INT PleaseShowFileMessage;

//#define MAX_XML_FILE_SIZE 10000
#define MAX_FILES_IN_DIR		20
//#define DIR_FILELIST_MAX_SIZE 1024

_LOCAL FILE2_RW_typ  *pFileRW ;

_LOCAL FILE2_RW_typ File_RW2;

_LOCAL UDINT pRec;
_LOCAL UDINT recLen;

_LOCAL plcstring _fileName[64];
//_LOCAL USINT load_after_save;
_LOCAL UDINT pos;
_LOCAL UINT indx;

USINT _CMD ;

char tempStr[64];

//////////////////
void _Open(FILE2_RW_typ *f);
void _Close(FILE2_RW_typ *f);
void _Create(FILE2_RW_typ *f);
void _Read(FILE2_RW_typ *f);
void _Write(FILE2_RW_typ *f);
void _Delete(FILE2_RW_typ *f);
void _ReadDir(FILE2_RW_typ *f);
void _ReadFileInfo(FILE2_RW_typ *f);
void _Rename(FILE2_RW_typ *f);
void _Copy(FILE2_RW_typ *f);

//void DeleteExtension(char *p);

#endif
```

### Program Logical/ESAB (ANSIC)

#### ESAB_PS.c - Init, cyclic, exit code
```c
#include <bur/plctypes.h>

#ifdef _DEFAULT_INCLUDES
	#include <AsDefault.h>
#endif

#include <..\GlobalDef.h>
#include <..\GlobalDecl.h>
#include <..\Lib\LoggerLib.c>

#include <..\Lib\libUDP\libUDP.h>
#include <..\Lib\libUDP\libUDP.c>

#define REC_BUF_LEN 160

_LOCAL plcstring send_data[32];
_LOCAL USINT receive_data[REC_BUF_LEN];
//_LOCAL USINT temp_data[REC_BUF_LEN * 3];

_LOCAL UDP_typ2 ESAB_UDP;

_LOCAL USINT ESAB_Com_Step;

_LOCAL char ESAB_IP_Address[16];
_LOCAL char PLC_IP_Address[16];

////////////////////////////////////////////

//UDP Receive Callback function to push data on ring buffer
static void udpReceivedNewData(UDINT pRxBuffer, UDINT RxDataLen , UDINT ringBuf){

	//DBG("New Data Received  of Length %d \r\n" , RxDataLen);

	//ckConvertByteStreamToHex(pRxBuffer, temp_data, RxDataLen, sizeof(temp_data));
	//LogTxt(&LogMgr, "<< %s" , temp_data);
	//DBG("(Hex): %s  \r\n" , temp_data);

}
//UDP Transmit Callback function for debugging purpose
static void udpTransmitedNewData(UDINT pTxBuffer, UDINT pTxDataLen){

	//DBG("New Data Trasmitted of Length %d  \r\n " , pTxDataLen );
	//ckConvertByteStreamToHex(pTxBuffer, temp_data, pTxDataLen, sizeof(temp_data));
	//LogTxt(&LogMgr, ">> %s" , temp_data);
	//DBG("(Hex): %s  \r\n" , temp_data);

}

void Convert_UINT2HEX( char* txt, UINT inp);
void Convert_USINT2HEX( char* txt, USINT inp);
USINT  Convert_HEX2USINT(char* txt);
UINT  Convert_HEX2UINT(char* txt);

//_LOCAL TON_typ ESAB_Tmr;

void _INIT ProgramInit(void){
UDP_typ2 *udp;

	strcpy(ESAB_IP_Address , "192.168.10.205" );

	strcpy(PLC_IP_Address , "192.168.10.123" ); // My PLC  Address

	udp = &ESAB_UDP;

	udp->listener_config.port = 10001;
	udp->listener_config.buffer = receive_data;
	udp->listener_config.bufferSize = REC_BUF_LEN;
	udp->listener.iRxCallback = (UDINT)udpReceivedNewData;
	//udp->listener.iRxRingBuf = (UDINT)&RingBufIn;

	udp->send.iPort = 10001;
	udp->send.iBuffer = send_data;
	udp->send.iBufferSize = REC_BUF_LEN;
	udp->send.iTxCallback = (UDINT)udpTransmitedNewData;

	strcpy(udp->send.iIPaddress , ESAB_IP_Address);
	udp->internal.UdpOpen_0.pIfAddr = (UDINT)&PLC_IP_Address[0];

	ESAB_PS.step = 0;

	ESAB_PS.Msc.Main_Tmr.PT = 1000;
	ESAB_PS.Msc.Cmd_Hrbt_Tmr.PT = 400;

	//ESAB_Tmr.PT = 1000;

	ESAB_PS.step = 1;

}

void _CYCLIC ProgramCyclic(void){
ESAB_typ *esab;
UDP_typ2 *udp;

USINT  status;
INT myINT;

	esab = &ESAB_PS;
	udp = &ESAB_UDP;

	Udp_cyclic(udp);

	switch(esab->step){

		case 0: // Wait

		break;

		case 1:

			if(udp->internal.step == 5){

				esab->Msc._voltage = esab->Param.Voltage;
				esab->Msc._amps = esab->Param.Amps;

				esab->Cmd.QuickStop = 0;
				esab->Cmd.WeldON = 0;

				esab->Msc._quickStop = esab->Cmd.QuickStop;
				esab->Msc._weldON = esab->Cmd.WeldON;

				strcpy (send_data , "R.001");
				udp->send.iBufferSize = 5;
				udp->send.iSendCMD = 1;

				esab->Msc.Main_Tmr.IN = 0;
				TON(&esab->Msc.Main_Tmr);
				esab->Msc.Main_Tmr.IN = 1;

				esab->Msc.Cmd_Hrbt_Tmr.IN = 0;
				TON(&esab->Msc.Cmd_Hrbt_Tmr);
				esab->Msc.Cmd_Hrbt_Tmr.IN = 1;

				esab->Msc._recev_counts  =	udp->listener.oStatus.counts;
				esab->step ++;

			}

		break;

		case 2:

			if(esab->Msc._recev_counts  !=  udp->listener.oStatus.counts){

				esab->Cmd.UpdateParam = 1;
				esab->step++;

			}
			else if(esab->Msc.Main_Tmr.Q)
				esab->step = 1;

		break;

		case 3:

			if(esab->Cmd.UpdateParam){
				esab->Cmd.UpdateParam = 0;

				esab->Msc._quickStop = !esab->Cmd.QuickStop;
				esab->Msc._weldON = !esab->Cmd.WeldON;
				esab->Msc._wF_Jog_FWD = !esab->Cmd.WF_Jog_FWD;
				esab->Msc._wF_Jog_REV = !esab->Cmd.WF_Jog_REV;
				esab->Msc._inputArea = !esab->Cmd.InputArea;
				esab->Msc._jogHighSpeed = !esab->Cmd.JogHighSpeed;

				esab->Msc._regulType = esab->Param.RegulType + 1;
				esab->Msc._voltage = esab->Param.Voltage + 1.0;
				esab->Msc._amps = esab->Param.Amps + 1.0;

			}

			if(esab->Msc.Cmd_Hrbt_Tmr.Q){
				//&& (!esab->Cmd.QuickStop)){

				strcpy(send_data , "W.001.000.008=0000000000000000");
				//strcpy(send_data , "W.001.000.008=000000000000000000000");

				//////  Byte 0 - Command LSB
				status = 0;
				if(esab->Cmd.WeldON)
					status += 0x1;

				//if(esab->Cmd.QuickStop)
					//status += 0x2;

				if(esab->Cmd.WF_Jog_FWD)
					status += 0x10;

				if(esab->Cmd.WF_Jog_REV)
					status += 0x20;

				Convert_USINT2HEX(&send_data[14], status);

				//strcpy(send_data , "W.001.000.001=00");
				//Convert_USINT2HEX(&send_data[14], status);

				//// Byte 1 - Command MSB

				status = (esab->Cmd.JogHighSpeed)? 0x4:0;
				Convert_USINT2HEX(&send_data[16], status);

				//status = (esab->Cmd.JogHighSpeed)? 0x4:0;
				//strcpy(send_data , "W.001.001.001=00");
				//Convert_USINT2HEX(&send_data[14], status);

				//// Byte 7 - HeartBeat to ESAB
				Convert_USINT2HEX(&send_data[28], esab->Msc._heartBeat++);

				//strcpy(send_data , "W.001.007.001=00");
				//Convert_USINT2HEX(&send_data[14], esab->Msc._heartBeat++);

				///////////////////////////////////////////////////////

				ESAB_UDP.send.iBufferSize = 30;
				ESAB_UDP.send.iSendCMD = 1;

				esab->Msc.Main_Tmr.IN = 0;
				TON(&esab->Msc.Main_Tmr);
				esab->Msc.Main_Tmr.IN = 1;

				esab->step = 11;

				////////////////////////////////////////
				///////////////////////////////////////

				/*
				strcpy(send_data , "W.001.007.001=00");

				Convert_USINT2HEX(&send_data[14], esab->Msc._heartBeat++);

				ESAB_UDP.send.iBufferSize = 16;
				ESAB_UDP.send.iSendCMD = 1;

				esab->Msc.Main_Tmr.IN = 0;
				TON(&esab->Msc.Main_Tmr);
				esab->Msc.Main_Tmr.IN = 1;

				esab->step = 11;
				*/

			}

			else if((esab->Cmd.QuickStop != esab->Msc._quickStop)
				|| (esab->Cmd.WeldON != esab->Msc._weldON)
				 || (esab->Cmd.WF_Jog_FWD != esab->Msc._wF_Jog_FWD)
				 || (esab->Cmd.WF_Jog_REV != esab->Msc._wF_Jog_REV)
				 ){
			//else if(0){

				/*
				esab->Msc._quickStop = esab->Cmd.QuickStop;
				esab->Msc._weldON = esab->Cmd.WeldON;
				esab->Msc._wF_Jog_FWD = esab->Cmd.WF_Jog_FWD;
				esab->Msc._wF_Jog_REV = esab->Cmd.WF_Jog_REV;
				*/

				status = 0;
				if(esab->Cmd.WeldON)
					status += 0x1;

				//if(esab->Cmd.QuickStop)
					//status += 0x2;

				if(esab->Cmd.WF_Jog_FWD)
					status += 0x10;

				if(esab->Cmd.WF_Jog_REV)
					status += 0x20;

				strcpy(send_data , "W.001.000.001=00");

				Convert_USINT2HEX(&send_data[14], status);

				ESAB_UDP.send.iBufferSize = 16;
				ESAB_UDP.send.iSendCMD = 1;

				esab->Msc.Main_Tmr.IN = 0;
				TON(&esab->Msc.Main_Tmr);
				esab->Msc.Main_Tmr.IN = 1;

				esab->step = 10;

			}
			/*
			else if(esab->Cmd.InputArea != esab->Msc._inputArea){
				esab->Msc._inputArea = esab->Cmd.InputArea;

				strcpy(send_data , "W.001.003.001=00");

				status = 0;
				if(esab->Cmd.InputArea)
					status += 0x4;

				Convert_USINT2HEX(&send_data[14], status);

				ESAB_UDP.send.iBufferSize = 16;
				ESAB_UDP.send.iSendCMD = 1;

				esab->Msc.Main_Tmr.IN = 0;
				TON(&esab->Msc.Main_Tmr);
				esab->Msc.Main_Tmr.IN = 1;

				esab->step = 10;

			}
			else if(esab->Param.RegulType != esab->Msc._regulType){
				esab->Msc._regulType = esab->Param.RegulType;

				strcpy(send_data , "W.001.009.001=00");

				Convert_USINT2HEX(&send_data[14], esab->Param.RegulType);

				ESAB_UDP.send.iBufferSize = 16;
				ESAB_UDP.send.iSendCMD = 1;

				esab->Msc.Main_Tmr.IN = 0;
				TON(&esab->Msc.Main_Tmr);
				esab->Msc.Main_Tmr.IN = 1;

				esab->step = 10;

			}
			*/
			else if(esab->Param.Voltage != esab->Msc._voltage){
				esab->Msc._voltage = esab->Param.Voltage;

				strcpy (send_data , "W.001.010.002=0000");

				Convert_UINT2HEX(&send_data[14], (esab->Param.Voltage * 10.0));

				ESAB_UDP.send.iBufferSize = 18;
				ESAB_UDP.send.iSendCMD = 1;

				esab->Msc.Main_Tmr.IN = 0;
				TON(&esab->Msc.Main_Tmr);
				esab->Msc.Main_Tmr.IN = 1;

				esab->step = 10;

			}
			else if(esab->Param.Amps != esab->Msc._amps){
				esab->Msc._amps = esab->Param.Amps;

				strcpy (send_data , "W.001.014.002=0000");

				Convert_UINT2HEX(&send_data[14], esab->Param.Amps);

				ESAB_UDP.send.iBufferSize = 18;
				ESAB_UDP.send.iSendCMD = 1;

				esab->Msc.Main_Tmr.IN = 0;
				TON(&esab->Msc.Main_Tmr);
				esab->Msc.Main_Tmr.IN = 1;

				esab->step = 10;

			}
			else if(esab->Cmd.JogHighSpeed != esab->Msc._jogHighSpeed){
				esab->Msc._jogHighSpeed = esab->Cmd.JogHighSpeed;

				status = (esab->Cmd.JogHighSpeed)? 0x4:0;

				strcpy(send_data , "W.001.001.001=00");

				Convert_USINT2HEX(&send_data[14], status);

				ESAB_UDP.send.iBufferSize = 16;
				ESAB_UDP.send.iSendCMD = 1;

				esab->Msc.Main_Tmr.IN = 0;
				TON(&esab->Msc.Main_Tmr);
				esab->Msc.Main_Tmr.IN = 1;

				esab->step = 10;

			}
			else{

				strcpy (send_data , "R.001");
				udp->send.iBufferSize = 5;
				udp->send.iSendCMD = 1;

				esab->Msc.Main_Tmr.IN = 0;
				TON(&esab->Msc.Main_Tmr);
				esab->Msc.Main_Tmr.IN = 1;

				esab->step = 50;
			}

		break;

		case 10: // Wait and Parse for Responde

			if(esab->Msc._recev_counts  !=  udp->listener.oStatus.counts){
				esab->Msc._recev_counts  ==  udp->listener.oStatus.counts;

				esab->Msc._quickStop = esab->Cmd.QuickStop;
				esab->Msc._weldON = esab->Cmd.WeldON;
				esab->Msc._wF_Jog_FWD = esab->Cmd.WF_Jog_FWD;
				esab->Msc._wF_Jog_REV = esab->Cmd.WF_Jog_REV;

				//esab->step = 0;
				esab->step = 3;

			}else if(esab->Msc.Main_Tmr.Q){
				ESAB_Tmo_Err = 1;
				esab->step = 1;

			}

		break;

		case 11: // Wait and Parse for Responde -  Command HeartBeat

			if(esab->Msc._recev_counts  !=  udp->listener.oStatus.counts){
				esab->Msc._recev_counts  ==  udp->listener.oStatus.counts;

				esab->Msc.Cmd_Hrbt_Tmr.IN = 0;
				TON(&esab->Msc.Cmd_Hrbt_Tmr);
				esab->Msc.Cmd_Hrbt_Tmr.IN = 1;

				//esab->step = 0;
				esab->step = 3;

			}else if(esab->Msc.Main_Tmr.Q){
				ESAB_Tmo_Err = 2;
				esab->step = 1;
			}

		break;

		case 50: // Parse Fbk

			if(esab->Msc._recev_counts  !=  udp->listener.oStatus.counts){

				//// Nowe

				// Sprawdzone
				status = Convert_HEX2USINT(&receive_data[2]);
				//esab->Fbk.Status = status & 0x07;
				esab->Fbk.Status = status;
				esab->Fbk.Error = (status & 0x8)? 1:0;

				status = Convert_HEX2USINT(&receive_data[4]);
				esab->Fbk.StatusMSB = status;
				esab->Fbk.ReadyToStart = (status & 0x8)? 1:0;

				status = Convert_HEX2USINT(&receive_data[8]);
				esab->Fbk.InputAreaActive = (status & 0x4)? 1:0;

				esab->Fbk.ErrorNum = Convert_HEX2USINT(&receive_data[10]);

				esab->Fbk.actVolts = ((float)Convert_HEX2UINT(&receive_data[18]))/10.0;
				esab->Fbk.actAmps = ((float)Convert_HEX2UINT(&receive_data[22]));
				esab->Fbk.actHeat = ((float)Convert_HEX2UINT(&receive_data[26]));

				myINT = (INT)Convert_HEX2UINT(&receive_data[30]);
				esab->Fbk.actWF = (float)myINT;

				esab->Fbk.SetRegulType = Convert_HEX2USINT(&receive_data[40]);

				esab->Fbk.SetVoltage = ((float)Convert_HEX2UINT(&receive_data[50]))/10.0;
				esab->Fbk.SetAmps = ((float)Convert_HEX2UINT(&receive_data[54]));
				esab->Fbk.SetWF = ((float)Convert_HEX2UINT(&receive_data[58]));
				esab->Fbk.SetTVL = ((float)Convert_HEX2UINT(&receive_data[62]));

				myINT = (INT)Convert_HEX2UINT(&receive_data[14]);
				esab->Fbk.Req_TVL_Speed = (float)myINT;

				myINT = (INT)Convert_HEX2UINT(&receive_data[78]);
				esab->Fbk.Req_WF_Speed = (float)myINT;

				esab->Fbk.ErrorCode = Convert_HEX2UINT(&receive_data[82]);
				esab->Fbk.ErrorSubCode = Convert_HEX2USINT(&receive_data[86]);
				esab->Fbk.ErrorNodeID = Convert_HEX2USINT(&receive_data[88]);

				esab->Fbk.HeartBeat = Convert_HEX2UINT(&receive_data[94]);

				if(esab->Fbk.ErrorNum != 0){
					if(esab->Fbk.ErrorNum != esab->Msc._errorNum){
						esab->Msc._errorNum = esab->Fbk.ErrorNum;
						esab->Fbk.NewErrorCode = esab->Fbk.ErrorCode;
					}
				}

				esab->Msc._recev_counts  =  udp->listener.oStatus.counts;

				//esab->step = 0;
				esab->step = 3;
			}
			else if(esab->Msc.Main_Tmr.Q){
				ESAB_Tmo_Err = 3;
				esab->step = 1;
			}

		break;

	}

	TON(&esab->Msc.Main_Tmr);
	TON(&esab->Msc.Cmd_Hrbt_Tmr);

}

void Convert_UINT2HEX( char* txt, UINT inp){
USINT val[4];
char *str;
str = "0123456789ABCDEF";

		val[0] = (USINT)(inp/(256*16));
		val[1] = (USINT)(inp/256%16);
		val[2] = (USINT)(inp%256/16);
		val[3] = (USINT)(inp%256%16);

		txt[2] = str[val[0]];
		txt[3] = str[val[1]];
		txt[0] = str[val[2]];
		txt[1] = str[val[3]];

}
void Convert_USINT2HEX( char* txt, USINT inp){
USINT val[2];
char *str;
str = "0123456789ABCDEF";

		val[0] = (USINT)(inp/16);
		val[1] = (USINT)(inp%16);

		txt[0] = str[val[0]];
		txt[1] = str[val[1]];

}

USINT  Convert_HEX2USINT(char* txt){
USINT ret = 0;

		if(txt[0] >= 'a')
			ret =((USINT)txt[0] - 'a' + 10)  * 16;
		else if(txt[0] >= 'A')
			ret = ((USINT)txt[0] - 'A' + 10) * 16;
		else if(txt[0] >= '0')
			ret =((USINT)txt[0] - '0') * 16;

		if(txt[1] >= 'a')
			ret +=(USINT)txt[1] - 'a' + 10;
		else if(txt[1] >= 'A')
			ret +=(USINT)txt[1] - 'A' +10;
		else if(txt[1] >= '0')
			ret +=((USINT)txt[1] - '0');

	return ret;

}

UINT  Convert_HEX2UINT(char* txt){
UINT ret = 0;
UINT ret2 = 0;

		if(txt[0] >= 'a')
			ret =((USINT)txt[0] - 'a' + 10)  * 16;
		else if(txt[0] >= 'A')
			ret = ((USINT)txt[0] - 'A' + 10) * 16;
		else if(txt[0] >= '0')
			ret =((USINT)txt[0] - '0') * 16;

		if(txt[1] >= 'a')
			ret +=(USINT)txt[1] - 'a' + 10;
		else if(txt[1] >= 'A')
			ret +=(USINT)txt[1] - 'A' +10;
		else if(txt[1] >= '0')
			ret +=((USINT)txt[1] - '0');

		if(txt[2] >= 'a')
			ret2 =((USINT)txt[2] - 'a' + 10)  * 16;
		else if(txt[2] >= 'A')
			ret2 = ((USINT)txt[2] - 'A' + 10) * 16;
		else if(txt[2] >= '0')
			ret2 =((USINT)txt[2] - '0') * 16;

		if(txt[3] >= 'a')
			ret2 +=((USINT)txt[3] - 'a' + 10);
		else if(txt[3] >= 'A')
			ret2 +=((USINT)txt[3] - 'A' +10);
		else if(txt[3] >= '0')
			ret2 +=((USINT)txt[3] - '0');

	return ret  + ret2  * 256;

}

void ckConvertByteStreamToHex(USINT* in , USINT* out , int lenIn , int lenOut ){
int i , ii , k;
char *str;
USINT val;

	str = "0123456789ABCDEF";

	for (i = 0 ; i < lenIn ; i++){

			val = in[i];

			for(k = 1 ; k >=0 ; k-- ){

				ii = k+ i*3;

				if(ii < lenOut){
					out[ii] = str[val % 16];
					val /= 16;
				}
				else {

					out[ii - 1] = 0;
					return;

				}

			}

			ii = 2 + i*3;

			if(ii < lenOut)
				out[ii] = ' ';
			else{

				out[ii - 1] = 0;
				return;

			}

		}

		ii++;

		if(ii < lenOut)
			out[ii] = 0;
		else
			out[ii - 1] = 0;

}
```

### statelib.c
```c
/*********************************************************
* FILE    	: 		statelib.c
*
* OBJECT	: 	N/A
*
* OVERVIEW	: 	Common Prototypes and Dependancies
*
*
* HISTORY : 		02.20.06 - Version 1
*
*
*
*
* DEPENDANCIES:
*********************************************************/

#ifndef _STATELIB_C
#define _STATELIB_C

#include <..\lib\WSI_types.h>

#include <..\lib\statelib.h>
//#include <string.h>
#include <..\lib\xstring.c>

/********************************************************
* CODE BASE:
*********************************************************/

plcbit SmTimerDone(struct SM_obj* sm){
	return sm->Tmr1.Q;
}
void SmTimerStart(struct SM_obj* sm, float timeoutTime){

	sm->Tmr1.IN = 0;
	TON(&sm->Tmr1);
	sm->Tmr1.IN = 1;
	sm->Tmr1.PT = (int) ((timeoutTime * 1000.0)+0.5);
	TON(&sm->Tmr1);

}

SINT HSReset( HS_obj *hs )
{
	memset( hs, 0, sizeof(HS_obj ));
	return 0;
}

BOOL HSCompare( HS_obj *hs, DINT status, DINT compare )
{
	/* Proper Execution: Upstream Process */
	if ( status == compare ) {
		hs->Ready	= 1;
		hs->Error	= 0;
		return 1;
	}
	else
		return 0;
}

DINT TimerStart( TON_typ *timer, REAL timeoutTime ) {
	timer->IN = 0;
	TON(timer);
	timer->IN = 1;
	timer->PT = (int) ((timeoutTime * 1000.0)+0.5);
	TON(timer);
	return 1;
}

BOOL TimerExecute( TON_typ *timer ) {
	TON(timer);
	return 1;
}

REAL TimerTimeRemaining( TON_typ *timer ) {
	return  ( (REAL) (timer->PT - timer->ET) /1000.0);
}

BOOL TimerIsTimeOut( TON_typ *timer ) {
	return timer->Q;
}

DINT sm_init( SM_obj *sm  )
{

	/* Text Field: */
	strcpy( sm->Text, "Yet to be Started" );

	/* Default */
	sm->oldStep			= 255;
	sm->Step			= 0;
	return 1;
}

DINT sm_serv( SM_obj *sm )
{
	/* Step Transition */
	if (sm->Step != sm->oldStep) {
		sm->new		= ON;
	    	sm->oldStep 		= sm->Step;
	}

	TimerExecute(&sm->Tmr1);
	return 1;
}

BOOL sm_reset( SM_obj *sm, BOOL Go )
{

	/* Bad Pointer or No New Data */
	if (sm == 0)
		return OFF;

	/* Default */
	sm->oldStep 		= 255;
	sm->Step			= 0;

	/* Return */
	return ON;
}

DINT sm_text( STRING text[32] , SM_obj *sm)
{
USINT stringh[50];

	/* Bad Pointer or No New Data */
	if ((sm == 0) || (!sm->new) )
		return 0;

	/* Turn Off Signal */
	sm->new = OFF;

	if(strlen(text)>31)
		xsprintf(sm->Text,"%d:%31s ", sm->Step , text );
	else
		xsprintf(sm->Text,"%d:%s", sm->Step , text );

	/* Check String Length */

	return 1;

}

UINT BitToWord( BOOL *b )
{
UINT i, wordh = 0;

	for (i=0;i<16;i++,b++)
		wordh = wordh + ((UINT) *b << i);

	return wordh;
}

/* Return: Quantity of High Bits */
USINT WordToBit( DINT x, BOOL *b)
{
UINT i;
USINT q = 0;

	/* Assign Masks */
	for (i=0;i<16;i++,b++) {
		*b = (BOOL) ( x >> i ) & 0x01;
		if (*b)
			q++;
	}

	return q;
}

UINT ToggleBit( UINT *wordh, UINT Bit_Num )
{
	if(Bit_Num >= 16)
		return *wordh;

	UINT offset = 1;
	offset <<= Bit_Num;

	if(*wordh & offset)
		ResetBit(wordh,Bit_Num );
	else
		SetBit(wordh,Bit_Num );

	return *wordh;
}

UINT SetBit( UINT *wordh, UINT Bit_Num )
{
UINT offset = 1;

	if(Bit_Num >= 16)
		return *wordh;

	offset <<= Bit_Num;

	*wordh |= (UINT) offset;

	return *wordh;
}
plcbit GetBit( UINT wordh, UINT Bit_Num )
{
UINT offset = 1;
plcbit ret;

	if(Bit_Num >= 16)
		return 0;

	offset <<= Bit_Num;

	ret = ((wordh & offset) > 0)? 1: 0;

	//return (plcbit)(wordh & offset);
	return ret;
}

UINT ResetBit( UINT *wordh, UINT Bit_Num )
{
UINT inverse = 0xFFFF;
UINT offset = 1;

	if(Bit_Num >= 16)
		return *wordh;

	offset <<= Bit_Num;

	inverse ^= offset;

	*wordh &= inverse;
	return *wordh;
}
//////
UDINT ToggleBit32( UDINT *wordh, UINT Bit_Num )
{
	if(Bit_Num >= 32)
		return *wordh;

	UDINT offset = 1;
	offset <<= Bit_Num;

	if(*wordh & offset)
		ResetBit32(wordh,Bit_Num );
	else
		SetBit32(wordh,Bit_Num );

	return *wordh;
}

UDINT SetBit32( UDINT *wordh, UINT Bit_Num )
{
UDINT offset = 1;

	if(Bit_Num >= 32)
		return *wordh;

	offset <<= Bit_Num;

	*wordh |= (UDINT) offset;

	return *wordh;
}
plcbit GetBit32( UDINT wordh, UINT Bit_Num )
{
UDINT offset = 1;

	if(Bit_Num >= 32)
		return 0;

	offset <<= Bit_Num;

	return (wordh & offset);
}

UDINT ResetBit32( UDINT *wordh, UINT Bit_Num )
{
UDINT inverse = 0xFFFF;
UDINT offset = 1;

	if(Bit_Num >= 32)
		return *wordh;

	offset <<= Bit_Num;

	inverse ^= offset;

	*wordh &= inverse;
	return *wordh;
}
//////

USINT GetHighBit( UINT wordh )
{
UINT Answer;
USINT i;

	for (i=0;i<16;i++) {
		Answer = (wordh >> i) & 0x0001;
		if (Answer > 0)
			return i;
	}
	return 0;
}

USINT GetNibble( USINT x, BOOL ho )
{
	if (ho) 	return ((x>>4)	& 0x0F);
	else		return ((x>>0)	& 0x0F);
}

USINT NibblesToByte(USINT o1, USINT o2)
{
	return (((o2<<4)  & 0xF0) | ((o1 & 0x0F)));
}
/* EOF */
#endif
```
